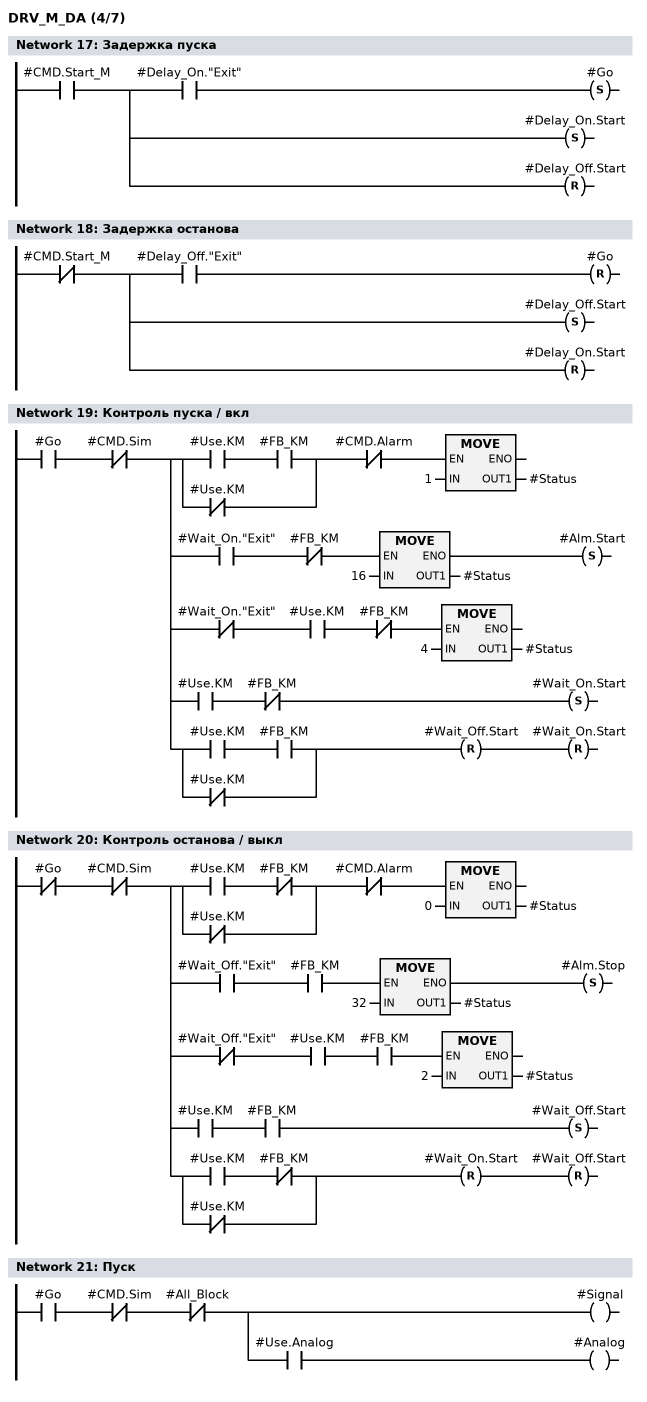
   RUNG wire#powerrail
      Contact( #CMD.Start_M )
      wire#w1
      Contact( #Delay_On."Exit" )
      S_Coil( #Go )
   END_RUNG
   RUNG wire#w1
      S_Coil( #Delay_On.Start )
   END_RUNG
   RUNG wire#w1
      R_Coil( #Delay_Off.Start )
   END_RUNG
   // the same network as SCL:
   IF #CMD.Start_M AND #Delay_On."Exit" THEN #Go := TRUE; END_IF;
   IF #CMD.Start_M THEN
       #Delay_On.Start := TRUE;
       #Delay_Off.Start := FALSE;
   END_IF;
END_REGION

REGION Network 18: Задержка останова
   RUNG wire#powerrail
      I_Contact( #CMD.Start_M )
      wire#w1
      Contact( #Delay_Off."Exit" )
      R_Coil( #Go )
   END_RUNG
   RUNG wire#w1
      S_Coil( #Delay_Off.Start )
   END_RUNG
   RUNG wire#w1
      R_Coil( #Delay_On.Start )
   END_RUNG
   // the same network as SCL:
   IF NOT #CMD.Start_M AND #Delay_Off."Exit" THEN #Go := FALSE; END_IF;
   IF NOT #CMD.Start_M THEN
       #Delay_Off.Start := TRUE;
       #Delay_On.Start := FALSE;
   END_IF;
END_REGION

REGION Network 19: Контроль пуска / вкл
   RUNG wire#powerrail
      Contact( #Go )
      I_Contact( #CMD.Sim )
      wire#w1
      Contact( #Use.KM )
      Contact( #FB_KM )
      wire#w2
      I_Contact( #CMD.Alarm )
      { S7_GenerateENO := "TRUE" } Move(in := 1, out1 => #Status)
   END_RUNG
   RUNG wire#w1
      I_Contact( #Use.KM )
   END_RUNG wire#w2
   RUNG wire#w1
      Contact( #Wait_On."Exit" )
      I_Contact( #FB_KM )
      { S7_GenerateENO := "TRUE" } Move(in := 16, out1 => #Status)
      S_Coil( #Alm.Start )
   END_RUNG
   RUNG wire#w1
      I_Contact( #Wait_On."Exit" )
      Contact( #Use.KM )
      I_Contact( #FB_KM )
      { S7_GenerateENO := "TRUE" } Move(in := 4, out1 => #Status)
   END_RUNG
   RUNG wire#w1
      Contact( #Use.KM )
      I_Contact( #FB_KM )
      S_Coil( #Wait_On.Start )
   END_RUNG
   RUNG wire#w1
      Contact( #Use.KM )
      Contact( #FB_KM )
      wire#w3
      R_Coil( #Wait_Off.Start )
      R_Coil( #Wait_On.Start )
   END_RUNG
   RUNG wire#w1
      I_Contact( #Use.KM )
   END_RUNG wire#w3
   // the same network as SCL:
   // ENO of a box is taken as its EN; it also drops when the box reports an error
   #_w1 := #Go AND NOT #CMD.Sim;
   IF #_w1 AND ((#Use.KM AND #FB_KM) OR NOT #Use.KM) AND NOT #CMD.Alarm THEN #Status := 1; END_IF;
   IF #_w1 AND #Wait_On."Exit" AND NOT #FB_KM THEN
       #Status := 16;
       #Alm.Start := TRUE;
   END_IF;
   IF #_w1 AND NOT #Wait_On."Exit" AND #Use.KM AND NOT #FB_KM THEN #Status := 4; END_IF;
   IF #_w1 AND #Use.KM AND NOT #FB_KM THEN #Wait_On.Start := TRUE; END_IF;
   IF #_w1 AND ((#Use.KM AND #FB_KM) OR NOT #Use.KM) THEN
       #Wait_Off.Start := FALSE;
       #Wait_On.Start := FALSE;
   END_IF;
END_REGION

REGION Network 20: Контроль останова / выкл
   RUNG wire#powerrail
      I_Contact( #Go )
      I_Contact( #CMD.Sim )
      wire#w1
      Contact( #Use.KM )
      I_Contact( #FB_KM )
      wire#w2
      I_Contact( #CMD.Alarm )
      { S7_GenerateENO := "TRUE" } Move(in := 0, out1 => #Status)
   END_RUNG
   RUNG wire#w1
      I_Contact( #Use.KM )
   END_RUNG wire#w2
   RUNG wire#w1
      Contact( #Wait_Off."Exit" )
      Contact( #FB_KM )
      { S7_GenerateENO := "TRUE" } Move(in := 32, out1 => #Status)
      S_Coil( #Alm.Stop )
   END_RUNG
   RUNG wire#w1
      I_Contact( #Wait_Off."Exit" )
      Contact( #Use.KM )
      Contact( #FB_KM )
      { S7_GenerateENO := "TRUE" } Move(in := 2, out1 => #Status)
   END_RUNG
   RUNG wire#w1
      Contact( #Use.KM )
      Contact( #FB_KM )
      S_Coil( #Wait_Off.Start )
   END_RUNG
   RUNG wire#w1
      Contact( #Use.KM )
      I_Contact( #FB_KM )
      wire#w3
      R_Coil( #Wait_On.Start )
      R_Coil( #Wait_Off.Start )
   END_RUNG
   RUNG wire#w1
      I_Contact( #Use.KM )
   END_RUNG wire#w3
   // the same network as SCL:
   // ENO of a box is taken as its EN; it also drops when the box reports an error
   #_w1 := NOT #Go AND NOT #CMD.Sim;
   IF #_w1 AND ((#Use.KM AND NOT #FB_KM) OR NOT #Use.KM) AND NOT #CMD.Alarm THEN #Status := 0; END_IF;
   IF #_w1 AND #Wait_Off."Exit" AND #FB_KM THEN
       #Status := 32;
       #Alm.Stop := TRUE;
   END_IF;
   IF #_w1 AND NOT #Wait_Off."Exit" AND #Use.KM AND #FB_KM THEN #Status := 2; END_IF;
   IF #_w1 AND #Use.KM AND #FB_KM THEN #Wait_Off.Start := TRUE; END_IF;
   IF #_w1 AND ((#Use.KM AND NOT #FB_KM) OR NOT #Use.KM) THEN
       #Wait_On.Start := FALSE;
       #Wait_Off.Start := FALSE;
   END_IF;
END_REGION

REGION Network 21: Пуск
   RUNG wire#powerrail
      Contact( #Go )
      I_Contact( #CMD.Sim )
      I_Contact( #All_Block )
      wire#w1
      Coil( #Signal )
   END_RUNG
   RUNG wire#w1
      Contact( #Use.Analog )
      Coil( #Analog )
   END_RUNG
   // the same network as SCL:
   #Signal := #Go AND NOT #CMD.Sim AND NOT #All_Block;
   #Analog := #Signal AND #Use.Analog;
END_REGION

REGION Network 22: Сервисный режим
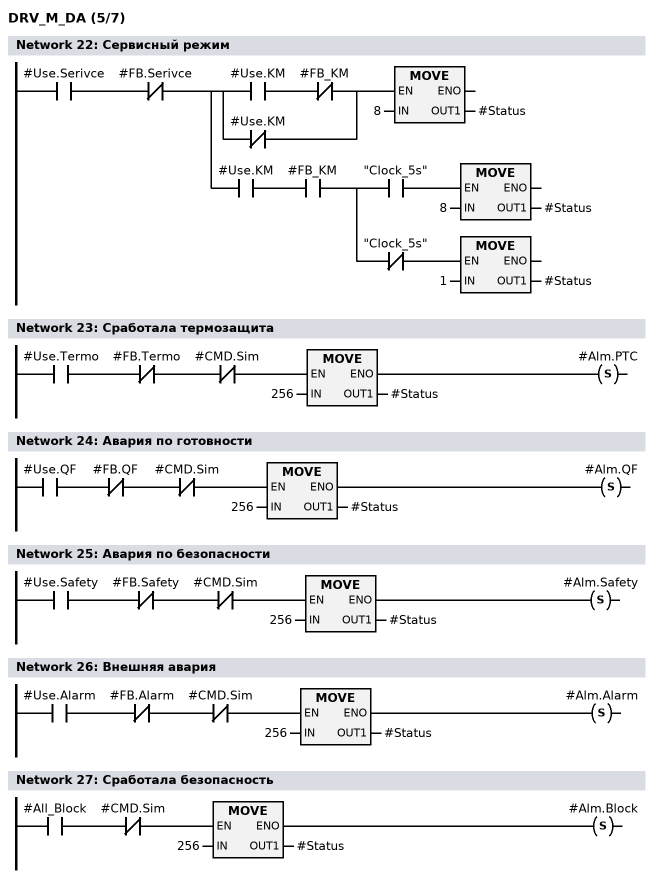
   RUNG wire#powerrail
      Contact( #Use.Serivce )
      I_Contact( #FB.Serivce )
      wire#w1
      Contact( #Use.KM )
      I_Contact( #FB_KM )
      wire#w2
      Move(in := 8, out1 => #Status)
   END_RUNG
   RUNG wire#w1
      I_Contact( #Use.KM )
   END_RUNG wire#w2
   RUNG wire#w1
      Contact( #Use.KM )
      Contact( #FB_KM )
      wire#w3
      Contact( "Clock_5s" )
      Move(in := 8, out1 => #Status)
   END_RUNG
   RUNG wire#w3
      I_Contact( "Clock_5s" )
      Move(in := 1, out1 => #Status)
   END_RUNG
   // the same network as SCL:
   #_w1 := #Use.Serivce AND NOT #FB.Serivce;
   IF #_w1 AND ((#Use.KM AND NOT #FB_KM) OR NOT #Use.KM) THEN #Status := 8; END_IF;
   #_w2 := #_w1 AND #Use.KM AND #FB_KM;
   IF #_w2 AND "Clock_5s" THEN #Status := 8; END_IF;
   IF #_w2 AND NOT "Clock_5s" THEN #Status := 1; END_IF;
END_REGION

REGION Network 23: Сработала термозащита
   RUNG wire#powerrail
      Contact( #Use.Termo )
      I_Contact( #FB.Termo )
      I_Contact( #CMD.Sim )
      { S7_GenerateENO := "TRUE" } Move(in := 256, out1 => #Status)
      S_Coil( #Alm.PTC )
   END_RUNG
   // the same network as SCL:
   // ENO of a box is taken as its EN; it also drops when the box reports an error
   IF #Use.Termo AND NOT #FB.Termo AND NOT #CMD.Sim THEN
       #Status := 256;
       #Alm.PTC := TRUE;
   END_IF;
END_REGION

REGION Network 24: Авария по готовности
   RUNG wire#powerrail
      Contact( #Use.QF )
      I_Contact( #FB.QF )
      I_Contact( #CMD.Sim )
      { S7_GenerateENO := "TRUE" } Move(in := 256, out1 => #Status)
      S_Coil( #Alm.QF )
   END_RUNG
   // the same network as SCL:
   // ENO of a box is taken as its EN; it also drops when the box reports an error
   IF #Use.QF AND NOT #FB.QF AND NOT #CMD.Sim THEN
       #Status := 256;
       #Alm.QF := TRUE;
   END_IF;
END_REGION

REGION Network 25: Авария по безопасности
   RUNG wire#powerrail
      Contact( #Use.Safety )
      I_Contact( #FB.Safety )
      I_Contact( #CMD.Sim )
      { S7_GenerateENO := "TRUE" } Move(in := 256, out1 => #Status)
      S_Coil( #Alm.Safety )
   END_RUNG
   // the same network as SCL:
   // ENO of a box is taken as its EN; it also drops when the box reports an error
   IF #Use.Safety AND NOT #FB.Safety AND NOT #CMD.Sim THEN
       #Status := 256;
       #Alm.Safety := TRUE;
   END_IF;
END_REGION

REGION Network 26: Внешняя авария
   RUNG wire#powerrail
      Contact( #Use.Alarm )
      I_Contact( #FB.Alarm )
      I_Contact( #CMD.Sim )
      { S7_GenerateENO := "TRUE" } Move(in := 256, out1 => #Status)
      S_Coil( #Alm.Alarm )
   END_RUNG
   // the same network as SCL:
   // ENO of a box is taken as its EN; it also drops when the box reports an error
   IF #Use.Alarm AND NOT #FB.Alarm AND NOT #CMD.Sim THEN
       #Status := 256;
       #Alm.Alarm := TRUE;
   END_IF;
END_REGION

REGION Network 27: Сработала безопасность
   RUNG wire#powerrail
      Contact( #All_Block )
      I_Contact( #CMD.Sim )
      { S7_GenerateENO := "TRUE" } Move(in := 256, out1 => #Status)
      S_Coil( #Alm.Block )
   END_RUNG
   // the same network as SCL:
   // ENO of a box is taken as its EN; it also drops when the box reports an error
   IF #All_Block AND NOT #CMD.Sim THEN
       #Status := 256;
       #Alm.Block := TRUE;
   END_IF;
END_REGION

REGION Network 28: Сигнал аварии
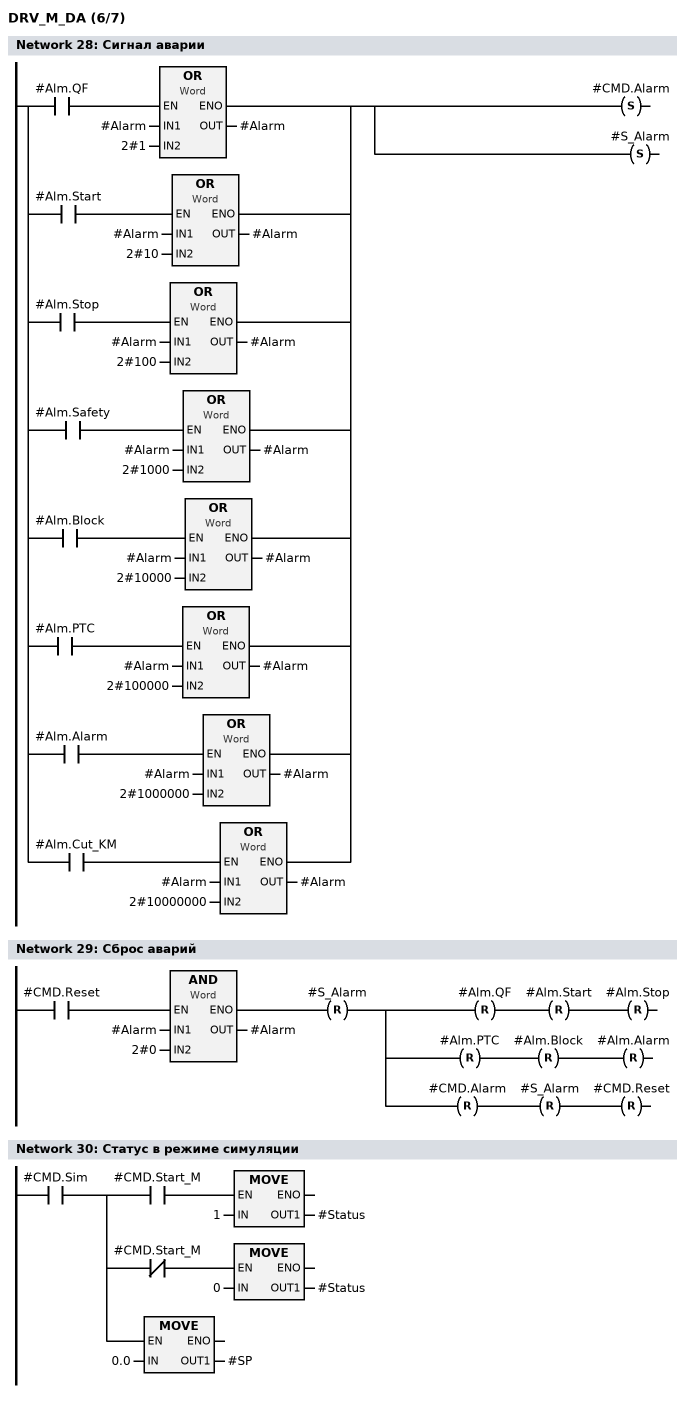
   // no checked SCL form for this network; see the picture
END_REGION

REGION Network 29: Сброс аварий
   // no checked SCL form for this network; see the picture
END_REGION

REGION Network 30: Статус в режиме симуляции
   RUNG wire#powerrail
      Contact( #CMD.Sim )
      wire#w1
      Contact( #CMD.Start_M )
      { S7_GenerateENO := "TRUE" } Move(in := 1, out1 => #Status)
   END_RUNG
   RUNG wire#w1
      I_Contact( #CMD.Start_M )
      { S7_GenerateENO := "TRUE" } Move(in := 0, out1 => #Status)
   END_RUNG
   RUNG wire#w1
      Move(in := 0.0, out1 => #SP)
   END_RUNG
   // the same network as SCL:
   IF #CMD.Sim AND #CMD.Start_M THEN #Status := 1; END_IF;
   IF #CMD.Sim AND NOT #CMD.Start_M THEN #Status := 0; END_IF;
   IF #CMD.Sim THEN #SP := 0.0; END_IF;
END_REGION

REGION Network 31: Статус в локальным режиме
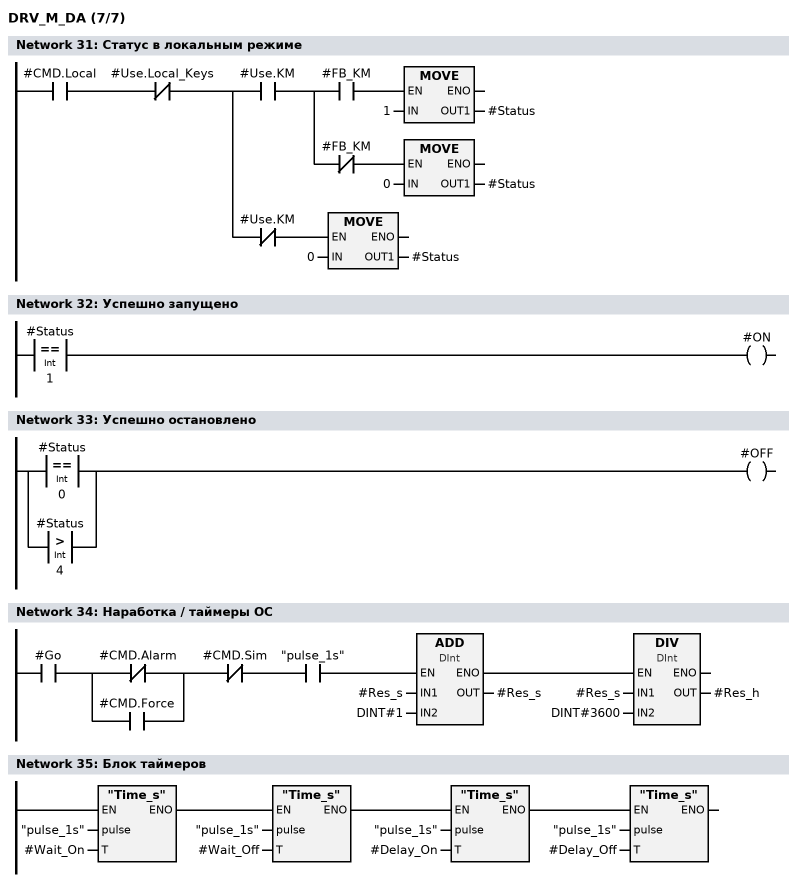
   RUNG wire#powerrail
      Contact( #CMD.Local )
      I_Contact( #Use.Local_Keys )
      wire#w1
      Contact( #Use.KM )
      wire#w2
      Contact( #FB_KM )
      { S7_GenerateENO := "TRUE" } Move(in := 1, out1 => #Status)
   END_RUNG
   RUNG wire#w2
      I_Contact( #FB_KM )
      { S7_GenerateENO := "TRUE" } Move(in := 0, out1 => #Status)
   END_RUNG
   RUNG wire#w1
      I_Contact( #Use.KM )
      { S7_GenerateENO := "TRUE" } Move(in := 0, out1 => #Status)
   END_RUNG
   // the same network as SCL:
   #_w1 := #CMD.Local AND NOT #Use.Local_Keys;
   #_w2 := #_w1 AND #Use.KM;
   IF #_w2 AND #FB_KM THEN #Status := 1; END_IF;
   IF #_w2 AND NOT #FB_KM THEN #Status := 0; END_IF;
   IF #_w1 AND NOT #Use.KM THEN #Status := 0; END_IF;
END_REGION

REGION Network 32: Успешно запущено
   RUNG wire#powerrail
      { S7_Templates := "SrcType := Int" } EQ_Contact(in1 := #Status, in2 := 1)
      Coil( #ON )
   END_RUNG
   // the same network as SCL:
   #ON := #Status = 1;
END_REGION

REGION Network 33: Успешно остановлено
   RUNG wire#powerrail
      { S7_Templates := "SrcType := Int" } EQ_Contact(in1 := #Status, in2 := 0)
      wire#w1
      Coil( #OFF )
   END_RUNG
   RUNG wire#powerrail
      { S7_Templates := "SrcType := Int" } GT_Contact(in1 := #Status, in2 := 4)
   END_RUNG wire#w1
   // the same network as SCL:
   #OFF := (#Status = 0) OR (#Status > 4);
END_REGION

REGION Network 34: Наработка / таймеры ОС
   RUNG wire#powerrail
      Contact( #Go )
      wire#w1
      I_Contact( #CMD.Alarm )
      wire#w2
      I_Contact( #CMD.Sim )
      Contact( "pulse_1s" )
      { S7_Templates := "SrcType := DInt"; S7_GenerateENO := "TRUE" } Add(in1 := #Res_s, in2 := DINT#1, out => #Res_s)
      { S7_Templates := "SrcType := DInt"; S7_GenerateENO := "TRUE" } Div(in1 := #Res_s, in2 := DINT#3600, out => #Res_h)
   END_RUNG
   RUNG wire#w1
      Contact( #CMD.Force )
   END_RUNG wire#w2
   // the same network as SCL:
   // ENO of a box is taken as its EN; it also drops when the box reports an error
   IF #Go AND (NOT #CMD.Alarm OR #CMD.Force) AND NOT #CMD.Sim AND "pulse_1s" THEN
       #Res_s := #Res_s + DINT#1;
       #Res_h := #Res_s / DINT#3600;
   END_IF;
END_REGION

REGION Network 35: Блок таймеров
   RUNG wire#powerrail
      "Time_s"(pulse := "pulse_1s", T := #Wait_On)
      "Time_s"(pulse := "pulse_1s", T := #Wait_Off)
      "Time_s"(pulse := "pulse_1s", T := #Delay_On)
      "Time_s"(pulse := "pulse_1s", T := #Delay_Off)
   END_RUNG
   // the same network as SCL:
   "Time_s"(pulse := "pulse_1s", T := #Wait_On, ENO => #_w1);
   "Time_s"(EN := #_w1, pulse := "pulse_1s", T := #Wait_Off, ENO => #_w2);
   "Time_s"(EN := #_w2, pulse := "pulse_1s", T := #Delay_On, ENO => #_w3);
   IF #_w3 THEN "Time_s"(pulse := "pulse_1s", T := #Delay_Off); END_IF;
END_REGION
END_FUNCTION_BLOCK

FUNCTION_BLOCK "DRV_V_D2"   // FB112, LAD
{ S7_Optimized_Access := 'FALSE' }
VERSION : 0.1
   VAR_INPUT
      FB_QF : Bool;   // защитный автомат / Защитный автомат
      FB_KM_Open : Bool;   // Пускатель - открыть
      FB_KM_Close : Bool;   // Пускатель - закрыть
      FB_Service : Bool;   // авария частотника / Сервисный выключатель
      FB_Open : Bool;   // ОС - открыто
      FB_Close : Bool;   // ОС - закрыто
      Local_Open : Bool;   // Локальное открытие
      Local_Close : Bool;   // Локальное закрытие
      All_Block : Bool;   // Аварийный останов
   END_VAR
   VAR_OUTPUT
      CMD_Open : Bool;   // Команда - открыть
      CMD_Close : Bool;   // Команда - закрыть
   END_VAR
   VAR_IN_OUT
      S_Alarm : Bool;   // Наличие аварии
   END_VAR
   VAR
      CMD : Struct   // Основные команды / Блок команд
         Hand : Bool;   // 0 - авто, 1 - ручной / 0 - Авто, 1 - Ручной
         Start_A : Bool;   // Автозапуск / Запуск в авторежиме
         Start_M : Bool;   // Ручной - вперёд / Запуск в ручном режиме
         Force : Bool;   // Принудительный
         Lock : Bool;   // Блокировать / Блокировка
         Local : Bool;   // Локальный
         Service : Bool;   // Сервис
         Safety : Bool;   // Безопасность
         Alarm : Bool;   // Есть авария / Авария
         Reset : Bool;   // Сброс аварий
         Sim : Bool;   // Режим симуляции
      END_STRUCT;
      Mode : Int;   // Режим работы
      Status : Int;   // Статус устройства
      Use : Struct   // Функционал
         Ready : Bool := true;   // Готовность
         QF : Bool := true;   // Защитный автомат
         KM_Open : Bool := true;   // Пускатель - открыть
         KM_Close : Bool;   // Пускатель - закрыть
         Serivce : Bool;   // Сервисный выключатель
         Open : Bool := true;   // ОС - открыто
         Close : Bool;   // ОС - закрыто
         Local_Keys : Bool;   // Использовать локальное управление
         One_KM : Bool;   // Общий пускатель
         Electro : Bool;   // Электропривод
      END_STRUCT;
      FB : Struct   // Функционал
         Ready : Bool;   // Готовность к запуску
         QF : Bool;   // Защитный автомат
         KM_Open : Bool;   // Пускатель - открыть
         KM_Close : Bool;   // Пускатель - закрыть
         Serivce : Bool;   // Сервисный выключатель
         Open : Bool;   // ОС - открыто
         Close : Bool;   // ОС - закрыто
         Reserv : Bool;
         Local_Open : Bool;   // Локальное открытие
         Local_Close : Bool;   // Локальное закрытие
      END_STRUCT;
      Go : Bool;   // Запуск
      ON : Bool;   // Успешно запущено
      OFF : Bool;   // Успешно остановлено
      G_Sim_On : Bool;   // Глобальная симуляция - начать
      G_Sim_Off : Bool;   // Глобальная симуляция - завершить
      REQ_Open : Bool;   // Запрос на открытие
      REQ_Close : Bool;   // Запрос на закрытие
      Wait_On : Struct   // Ожидание ОС контактора / Время на запуск
         SP : Int := 4;
         Now : Int;
         "Exit" : Bool;
         Start : Bool;
         Pause : Bool;
         Reset : Bool;   // Сброс таймера
      END_STRUCT;
      Wait_Off : Struct   // Ожидание концевиков / Время на останов
         SP : Int := 4;
         Now : Int;
         "Exit" : Bool;
         Start : Bool;
         Pause : Bool;
         Reset : Bool;   // Сброс таймера
      END_STRUCT;
      Delay_On : Struct
         SP : Real;   // Уставка
         Now : Real;   // Текущий счёт
         One : Real := 0.1;   // Вес импульса
         Progress : Real;   // Прогресс выполнения
         "Exit" : Bool;   // Счёт завершён
         Start : Bool;   // Запуск
         Pause : Bool;   // Пауза
         Reset : Bool;   // Сброс счёта
         pos : Bool;   // Контроль фронта сигнала
      END_STRUCT;
      Delay_Off : Struct
         SP : Real;   // Уставка
         Now : Real;   // Текущий счёт
         One : Real := 0.1;   // Вес импульса
         Progress : Real;   // Прогресс выполнения
         "Exit" : Bool;   // Счёт завершён
         Start : Bool;   // Запуск
         Pause : Bool;   // Пауза
         Reset : Bool;   // Сброс счёта
         pos : Bool;   // Контроль фронта сигнала
      END_STRUCT;
      Inv : Struct   // Инверсия сигналов
         Reserv : Bool;
         QF : Bool;   // Защитный автомат
         KM_Open : Bool;   // Пускатель - открыть
         KM_Close : Bool;   // Пускатель - закрыть
         Serivce : Bool;   // Сервисный выключатель
         Open : Bool;   // ОС - открыто
         Close : Bool;   // ОС - закрыто
         CMD : Bool;   // Инверсия управляющих сигналов
         Local_Open : Bool;   // Локальное открытие
         Local_Close : Bool;   // Локальное закрытие
      END_STRUCT;
      Alm : Struct   // Сбор аварий / Список аварий
         Block : Bool;   // Аварийная остановка
         QF : Bool;   // привод не готов / Выбило защитный автомат
         KM_Open : Bool;   // Не сработал пускатель - открыть
         KM_Close : Bool;   // Не сработал пускатель - закрыть
         Two_S : Bool;   // Две ОС
         Open : Bool;   // Не сработал концевик - открыто
         Close : Bool;   // термозащита / Не сработал концевик - закрыто
      END_STRUCT;
      Alarm : Word;   // Слово аварий
      Res_h : DInt;   // наработка (ч)
      Res_s : DInt;   // наработка (с)
      REQ_ON : "DRV_Micro";   // Контроль пускателя на открытие
      REQ_OFF : "DRV_Micro";   // Контроль пускателя на закрытие
   END_VAR
   VAR_TEMP   // added for the SCL form of the ladder/FBD networks
      _w1 : Bool;
      _w2 : Bool;
      _w3 : Bool;
   END_VAR
BEGIN

REGION Network 1: Режим глобальной симуляции
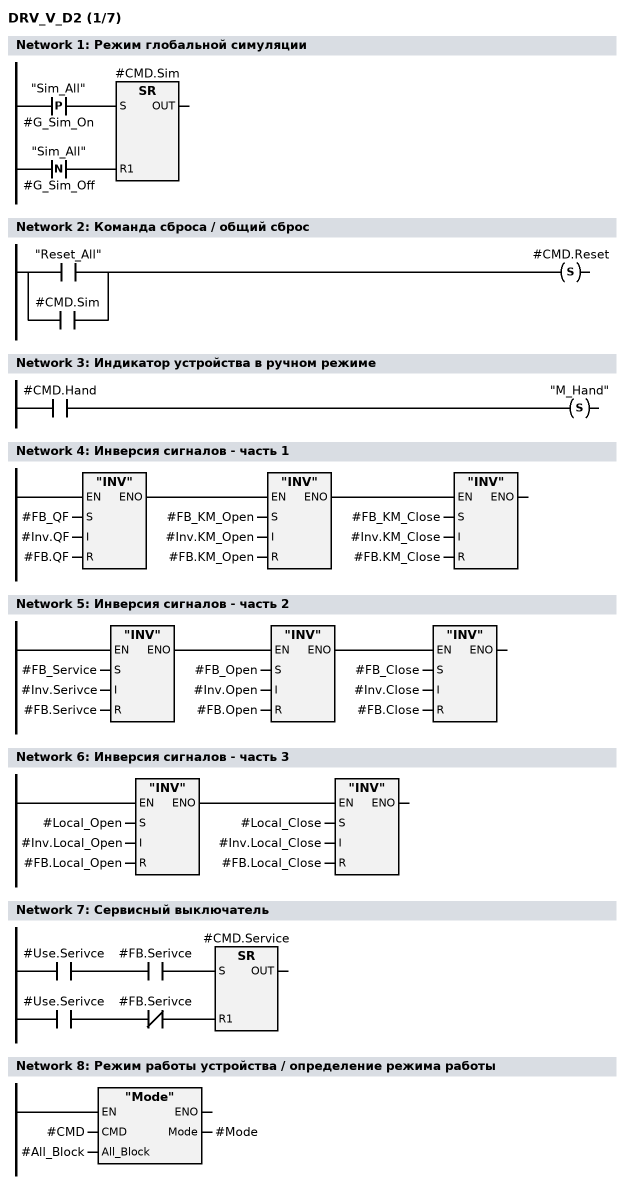
   RUNG wire#powerrail
      P_Contact(operand := "Sim_All", bit := #G_Sim_On)
      S_SR(operand := #CMD.Sim, r1 := wire#w1)
   END_RUNG
   RUNG wire#powerrail
      N_Contact(operand := "Sim_All", bit := #G_Sim_Off)
   END_RUNG wire#w1
   // the same network as SCL:
   #_w1 := "Sim_All" AND NOT #G_Sim_On;   // rising edge of "Sim_All"
   #G_Sim_On := "Sim_All";
   #_w2 := NOT "Sim_All" AND #G_Sim_Off;   // falling edge of "Sim_All"
   #G_Sim_Off := "Sim_All";
   IF #_w1 THEN
       #CMD.Sim := TRUE;   // SR flip-flop
   END_IF;
   IF #_w2 THEN #CMD.Sim := FALSE; END_IF;
END_REGION

REGION Network 2: Команда сброса / общий сброс
   RUNG wire#powerrail
      Contact( "Reset_All" )
      wire#w1
      S_Coil( #CMD.Reset )
   END_RUNG
   RUNG wire#powerrail
      Contact( #CMD.Sim )
   END_RUNG wire#w1
   // the same network as SCL:
   IF "Reset_All" OR #CMD.Sim THEN #CMD.Reset := TRUE; END_IF;
END_REGION

REGION Network 3: Индикатор устройства в ручном режиме
   RUNG wire#powerrail
      Contact( #CMD.Hand )
      S_Coil( "M_Hand" )
   END_RUNG
   // the same network as SCL:
   IF #CMD.Hand THEN "M_Hand" := TRUE; END_IF;
END_REGION

REGION Network 4: Инверсия сигналов - часть 1
   RUNG wire#powerrail
      "INV"(S := #FB_QF, I := #Inv.QF, R := #FB.QF)
      "INV"(S := #FB_KM_Open, I := #Inv.KM_Open, R := #FB.KM_Open)
      "INV"(S := #FB_KM_Close, I := #Inv.KM_Close, R := #FB.KM_Close)
   END_RUNG
   // the same network as SCL:
   "INV"(S := #FB_QF, I := #Inv.QF, R := #FB.QF, ENO => #_w1);
   "INV"(EN := #_w1, S := #FB_KM_Open, I := #Inv.KM_Open, R := #FB.KM_Open, ENO => #_w2);
   IF #_w2 THEN "INV"(S := #FB_KM_Close, I := #Inv.KM_Close, R := #FB.KM_Close); END_IF;
END_REGION

REGION Network 5: Инверсия сигналов - часть 2
   RUNG wire#powerrail
      "INV"(S := #FB_Service, I := #Inv.Serivce, R := #FB.Serivce)
      "INV"(S := #FB_Open, I := #Inv.Open, R := #FB.Open)
      "INV"(S := #FB_Close, I := #Inv.Close, R := #FB.Close)
   END_RUNG
   // the same network as SCL:
   "INV"(S := #FB_Service, I := #Inv.Serivce, R := #FB.Serivce, ENO => #_w1);
   "INV"(EN := #_w1, S := #FB_Open, I := #Inv.Open, R := #FB.Open, ENO => #_w2);
   IF #_w2 THEN "INV"(S := #FB_Close, I := #Inv.Close, R := #FB.Close); END_IF;
END_REGION

REGION Network 6: Инверсия сигналов - часть 3
   RUNG wire#powerrail
      "INV"(S := #Local_Open, I := #Inv.Local_Open, R := #FB.Local_Open)
      "INV"(S := #Local_Close, I := #Inv.Local_Close, R := #FB.Local_Close)
   END_RUNG
   // the same network as SCL:
   "INV"(S := #Local_Open, I := #Inv.Local_Open, R := #FB.Local_Open, ENO => #_w1);
   IF #_w1 THEN "INV"(S := #Local_Close, I := #Inv.Local_Close, R := #FB.Local_Close); END_IF;
END_REGION

REGION Network 7: Сервисный выключатель
   RUNG wire#powerrail
      Contact( #Use.Serivce )
      Contact( #FB.Serivce )
      S_SR(operand := #CMD.Service, r1 := wire#w1)
   END_RUNG
   RUNG wire#powerrail
      Contact( #Use.Serivce )
      I_Contact( #FB.Serivce )
   END_RUNG wire#w1
   // the same network as SCL:
   IF #Use.Serivce AND #FB.Serivce THEN
       #CMD.Service := TRUE;   // SR flip-flop
   END_IF;
   IF #Use.Serivce AND NOT #FB.Serivce THEN #CMD.Service := FALSE; END_IF;
END_REGION

REGION Network 8: Режим работы устройства / определение режима работы
   RUNG wire#powerrail
      "Mode"(CMD := #CMD, All_Block := #All_Block, Mode => #Mode)
   END_RUNG
   // the same network as SCL:
   "Mode"(CMD := #CMD, All_Block := #All_Block, Mode => #Mode);
END_REGION

REGION Network 9: Готовность к запуску
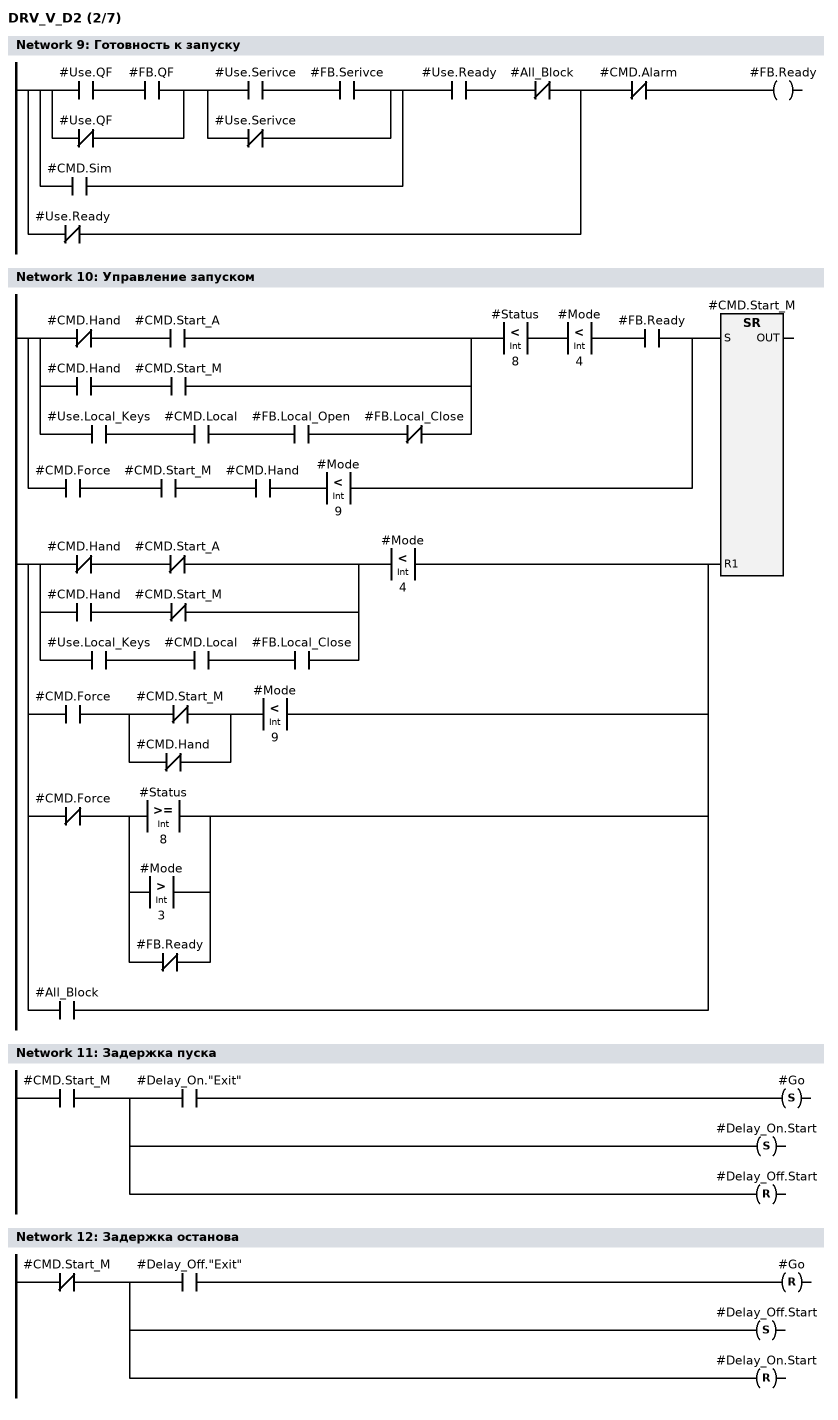
   RUNG wire#powerrail
      Contact( #Use.QF )
      Contact( #FB.QF )
      wire#w1
      Contact( #Use.Serivce )
      Contact( #FB.Serivce )
      wire#w2
      Contact( #Use.Ready )
      I_Contact( #All_Block )
      wire#w3
      I_Contact( #CMD.Alarm )
      Coil( #FB.Ready )
   END_RUNG
   RUNG wire#powerrail
      I_Contact( #Use.QF )
   END_RUNG wire#w1
   RUNG wire#w1
      I_Contact( #Use.Serivce )
   END_RUNG wire#w2
   RUNG wire#powerrail
      Contact( #CMD.Sim )
   END_RUNG wire#w2
   RUNG wire#powerrail
      I_Contact( #Use.Ready )
   END_RUNG wire#w3
   // the same network as SCL:
   #FB.Ready := ((((((#Use.QF AND #FB.QF) OR NOT #Use.QF) AND ((#Use.Serivce AND #FB.Serivce) OR NOT #Use.Serivce)) OR #CMD.Sim) AND #Use.Ready AND NOT #All_Block) OR NOT #Use.Ready) AND NOT #CMD.Alarm;
END_REGION

REGION Network 10: Управление запуском
   RUNG wire#powerrail
      I_Contact( #CMD.Hand )
      Contact( #CMD.Start_A )
      wire#w1
      { S7_Templates := "SrcType := Int" } LT_Contact(in1 := #Status, in2 := 8)
      { S7_Templates := "SrcType := Int" } LT_Contact(in1 := #Mode, in2 := 4)
      Contact( #FB.Ready )
      wire#w2
      S_SR(operand := #CMD.Start_M, r1 := wire#w7)
   END_RUNG
   RUNG wire#powerrail
      Contact( #CMD.Hand )
      Contact( #CMD.Start_M )
   END_RUNG wire#w1
   RUNG wire#powerrail
      Contact( #Use.Local_Keys )
      Contact( #CMD.Local )
      Contact( #FB.Local_Open )
      I_Contact( #FB.Local_Close )
   END_RUNG wire#w1
   RUNG wire#powerrail
      Contact( #CMD.Force )
      Contact( #CMD.Start_M )
      Contact( #CMD.Hand )
      { S7_Templates := "SrcType := Int" } LT_Contact(in1 := #Mode, in2 := 9)
   END_RUNG wire#w2
   RUNG wire#powerrail
      I_Contact( #CMD.Hand )
      I_Contact( #CMD.Start_A )
      wire#w3
      { S7_Templates := "SrcType := Int" } LT_Contact(in1 := #Mode, in2 := 4)
   END_RUNG wire#w7
   RUNG wire#powerrail
      Contact( #CMD.Hand )
      I_Contact( #CMD.Start_M )
   END_RUNG wire#w3
   RUNG wire#powerrail
      Contact( #Use.Local_Keys )
      Contact( #CMD.Local )
      Contact( #FB.Local_Close )
   END_RUNG wire#w3
   RUNG wire#powerrail
      Contact( #CMD.Force )
      wire#w4
      I_Contact( #CMD.Start_M )
      wire#w5
      { S7_Templates := "SrcType := Int" } LT_Contact(in1 := #Mode, in2 := 9)
   END_RUNG wire#w7
   RUNG wire#w4
      I_Contact( #CMD.Hand )
   END_RUNG wire#w5
   RUNG wire#powerrail
      I_Contact( #CMD.Force )
      wire#w6
      { S7_Templates := "SrcType := Int" } GE_Contact(in1 := #Status, in2 := 8)
   END_RUNG wire#w7
   RUNG wire#w6
      { S7_Templates := "SrcType := Int" } GT_Contact(in1 := #Mode, in2 := 3)
   END_RUNG wire#w7
   RUNG wire#w6
      I_Contact( #FB.Ready )
   END_RUNG wire#w7
   RUNG wire#powerrail
      Contact( #All_Block )
   END_RUNG wire#w7
   // the same network as SCL:
   #_w1 := (((NOT #CMD.Hand AND NOT #CMD.Start_A) OR (#CMD.Hand AND NOT #CMD.Start_M) OR (#Use.Local_Keys AND #CMD.Local AND #FB.Local_Close)) AND (#Mode < 4)) OR (#CMD.Force AND (NOT #CMD.Start_M OR NOT #CMD.Hand) AND (#Mode < 9)) OR (NOT #CMD.Force AND ((#Status >= 8) OR (#Mode > 3) OR NOT #FB.Ready)) OR #All_Block;
   IF (((NOT #CMD.Hand AND #CMD.Start_A) OR (#CMD.Hand AND #CMD.Start_M) OR (#Use.Local_Keys AND #CMD.Local AND #FB.Local_Open AND NOT #FB.Local_Close)) AND (#Status < 8) AND (#Mode < 4) AND #FB.Ready) OR (#CMD.Force AND #CMD.Start_M AND #CMD.Hand AND (#Mode < 9)) THEN
       #CMD.Start_M := TRUE;   // SR flip-flop
   END_IF;
   IF #_w1 THEN #CMD.Start_M := FALSE; END_IF;
END_REGION

REGION Network 11: Задержка пуска
   RUNG wire#powerrail
      Contact( #CMD.Start_M )
      wire#w1
      Contact( #Delay_On."Exit" )
      S_Coil( #Go )
   END_RUNG
   RUNG wire#w1
      S_Coil( #Delay_On.Start )
   END_RUNG
   RUNG wire#w1
      R_Coil( #Delay_Off.Start )
   END_RUNG
   // the same network as SCL:
   IF #CMD.Start_M AND #Delay_On."Exit" THEN #Go := TRUE; END_IF;
   IF #CMD.Start_M THEN
       #Delay_On.Start := TRUE;
       #Delay_Off.Start := FALSE;
   END_IF;
END_REGION

REGION Network 12: Задержка останова
   RUNG wire#powerrail
      I_Contact( #CMD.Start_M )
      wire#w1
      Contact( #Delay_Off."Exit" )
      R_Coil( #Go )
   END_RUNG
   RUNG wire#w1
      S_Coil( #Delay_Off.Start )
   END_RUNG
   RUNG wire#w1
      R_Coil( #Delay_On.Start )
   END_RUNG
   // the same network as SCL:
   IF NOT #CMD.Start_M AND #Delay_Off."Exit" THEN #Go := FALSE; END_IF;
   IF NOT #CMD.Start_M THEN
       #Delay_Off.Start := TRUE;
       #Delay_On.Start := FALSE;
   END_IF;
END_REGION

REGION Network 13: Команда открытия / выкл
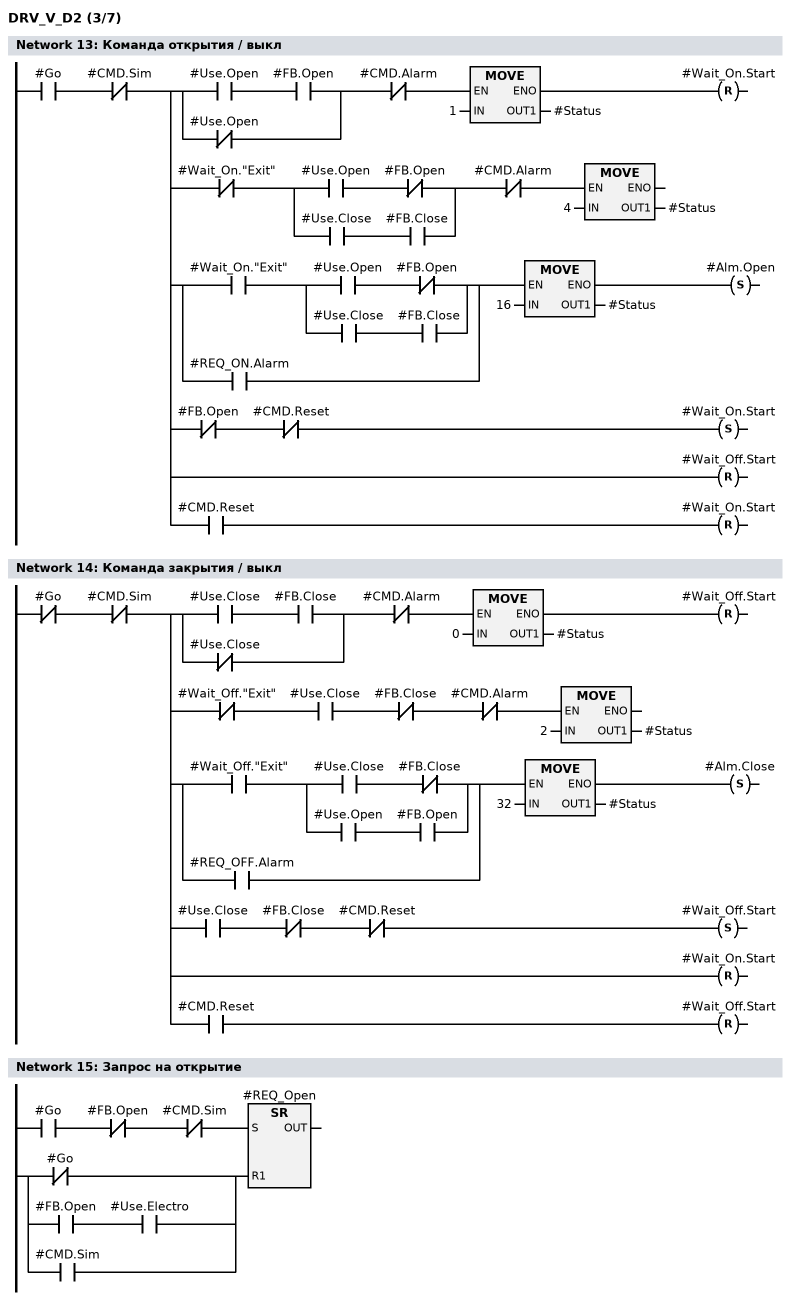
   RUNG wire#powerrail
      Contact( #Go )
      I_Contact( #CMD.Sim )
      wire#w1
      Contact( #Use.Open )
      Contact( #FB.Open )
      wire#w2
      I_Contact( #CMD.Alarm )
      { S7_GenerateENO := "TRUE" } Move(in := 1, out1 => #Status)
      R_Coil( #Wait_On.Start )
   END_RUNG
   RUNG wire#w1
      I_Contact( #Use.Open )
   END_RUNG wire#w2
   RUNG wire#w1
      I_Contact( #Wait_On."Exit" )
      wire#w3
      Contact( #Use.Open )
      I_Contact( #FB.Open )
      wire#w4
      I_Contact( #CMD.Alarm )
      { S7_GenerateENO := "TRUE" } Move(in := 4, out1 => #Status)
   END_RUNG
   RUNG wire#w3
      Contact( #Use.Close )
      Contact( #FB.Close )
   END_RUNG wire#w4
   RUNG wire#w1
      Contact( #Wait_On."Exit" )
      wire#w5
      Contact( #Use.Open )
      I_Contact( #FB.Open )
      wire#w6
      { S7_GenerateENO := "TRUE" } Move(in := 16, out1 => #Status)
      S_Coil( #Alm.Open )
   END_RUNG
   RUNG wire#w5
      Contact( #Use.Close )
      Contact( #FB.Close )
   END_RUNG wire#w6
   RUNG wire#w1
      Contact( #REQ_ON.Alarm )
   END_RUNG wire#w6
   RUNG wire#w1
      I_Contact( #FB.Open )
      I_Contact( #CMD.Reset )
      S_Coil( #Wait_On.Start )
   END_RUNG
   RUNG wire#w1
      R_Coil( #Wait_Off.Start )
   END_RUNG
   RUNG wire#w1
      Contact( #CMD.Reset )
      R_Coil( #Wait_On.Start )
   END_RUNG
   // the same network as SCL:
   // ENO of a box is taken as its EN; it also drops when the box reports an error
   #_w1 := #Go AND NOT #CMD.Sim;
   IF #_w1 AND ((#Use.Open AND #FB.Open) OR NOT #Use.Open) AND NOT #CMD.Alarm THEN
       #Status := 1;
       #Wait_On.Start := FALSE;
   END_IF;
   IF #_w1 AND NOT #Wait_On."Exit" AND ((#Use.Open AND NOT #FB.Open) OR (#Use.Close AND #FB.Close)) AND NOT #CMD.Alarm THEN
       #Status := 4;
   END_IF;
   IF #_w1 AND ((#Wait_On."Exit" AND ((#Use.Open AND NOT #FB.Open) OR (#Use.Close AND #FB.Close))) OR #REQ_ON.Alarm) THEN
       #Status := 16;
       #Alm.Open := TRUE;
   END_IF;
   IF #_w1 AND NOT #FB.Open AND NOT #CMD.Reset THEN #Wait_On.Start := TRUE; END_IF;
   IF #_w1 THEN #Wait_Off.Start := FALSE; END_IF;
   IF #_w1 AND #CMD.Reset THEN #Wait_On.Start := FALSE; END_IF;
END_REGION

REGION Network 14: Команда закрытия / выкл
   RUNG wire#powerrail
      I_Contact( #Go )
      I_Contact( #CMD.Sim )
      wire#w1
      Contact( #Use.Close )
      Contact( #FB.Close )
      wire#w2
      I_Contact( #CMD.Alarm )
      { S7_GenerateENO := "TRUE" } Move(in := 0, out1 => #Status)
      R_Coil( #Wait_Off.Start )
   END_RUNG
   RUNG wire#w1
      I_Contact( #Use.Close )
   END_RUNG wire#w2
   RUNG wire#w1
      I_Contact( #Wait_Off."Exit" )
      Contact( #Use.Close )
      I_Contact( #FB.Close )
      I_Contact( #CMD.Alarm )
      { S7_GenerateENO := "TRUE" } Move(in := 2, out1 => #Status)
   END_RUNG
   RUNG wire#w1
      Contact( #Wait_Off."Exit" )
      wire#w3
      Contact( #Use.Close )
      I_Contact( #FB.Close )
      wire#w4
      { S7_GenerateENO := "TRUE" } Move(in := 32, out1 => #Status)
      S_Coil( #Alm.Close )
   END_RUNG
   RUNG wire#w3
      Contact( #Use.Open )
      Contact( #FB.Open )
   END_RUNG wire#w4
   RUNG wire#w1
      Contact( #REQ_OFF.Alarm )
   END_RUNG wire#w4
   RUNG wire#w1
      Contact( #Use.Close )
      I_Contact( #FB.Close )
      I_Contact( #CMD.Reset )
      S_Coil( #Wait_Off.Start )
   END_RUNG
   RUNG wire#w1
      R_Coil( #Wait_On.Start )
   END_RUNG
   RUNG wire#w1
      Contact( #CMD.Reset )
      R_Coil( #Wait_Off.Start )
   END_RUNG
   // the same network as SCL:
   // ENO of a box is taken as its EN; it also drops when the box reports an error
   #_w1 := NOT #Go AND NOT #CMD.Sim;
   IF #_w1 AND ((#Use.Close AND #FB.Close) OR NOT #Use.Close) AND NOT #CMD.Alarm THEN
       #Status := 0;
       #Wait_Off.Start := FALSE;
   END_IF;
   IF #_w1 AND NOT #Wait_Off."Exit" AND #Use.Close AND NOT #FB.Close AND NOT #CMD.Alarm THEN
       #Status := 2;
   END_IF;
   IF #_w1 AND ((#Wait_Off."Exit" AND ((#Use.Close AND NOT #FB.Close) OR (#Use.Open AND #FB.Open))) OR #REQ_OFF.Alarm) THEN
       #Status := 32;
       #Alm.Close := TRUE;
   END_IF;
   IF #_w1 AND #Use.Close AND NOT #FB.Close AND NOT #CMD.Reset THEN #Wait_Off.Start := TRUE; END_IF;
   IF #_w1 THEN #Wait_On.Start := FALSE; END_IF;
   IF #_w1 AND #CMD.Reset THEN #Wait_Off.Start := FALSE; END_IF;
END_REGION

REGION Network 15: Запрос на открытие
   RUNG wire#powerrail
      Contact( #Go )
      I_Contact( #FB.Open )
      I_Contact( #CMD.Sim )
      S_SR(operand := #REQ_Open, r1 := wire#w1)
   END_RUNG
   RUNG wire#powerrail
      I_Contact( #Go )
   END_RUNG wire#w1
   RUNG wire#powerrail
      Contact( #FB.Open )
      Contact( #Use.Electro )
   END_RUNG wire#w1
   RUNG wire#powerrail
      Contact( #CMD.Sim )
   END_RUNG wire#w1
   // the same network as SCL:
   IF #Go AND NOT #FB.Open AND NOT #CMD.Sim THEN
       #REQ_Open := TRUE;   // SR flip-flop
   END_IF;
   IF NOT #Go OR (#FB.Open AND #Use.Electro) OR #CMD.Sim THEN #REQ_Open := FALSE; END_IF;
END_REGION

REGION Network 16: Запрос на закрытие
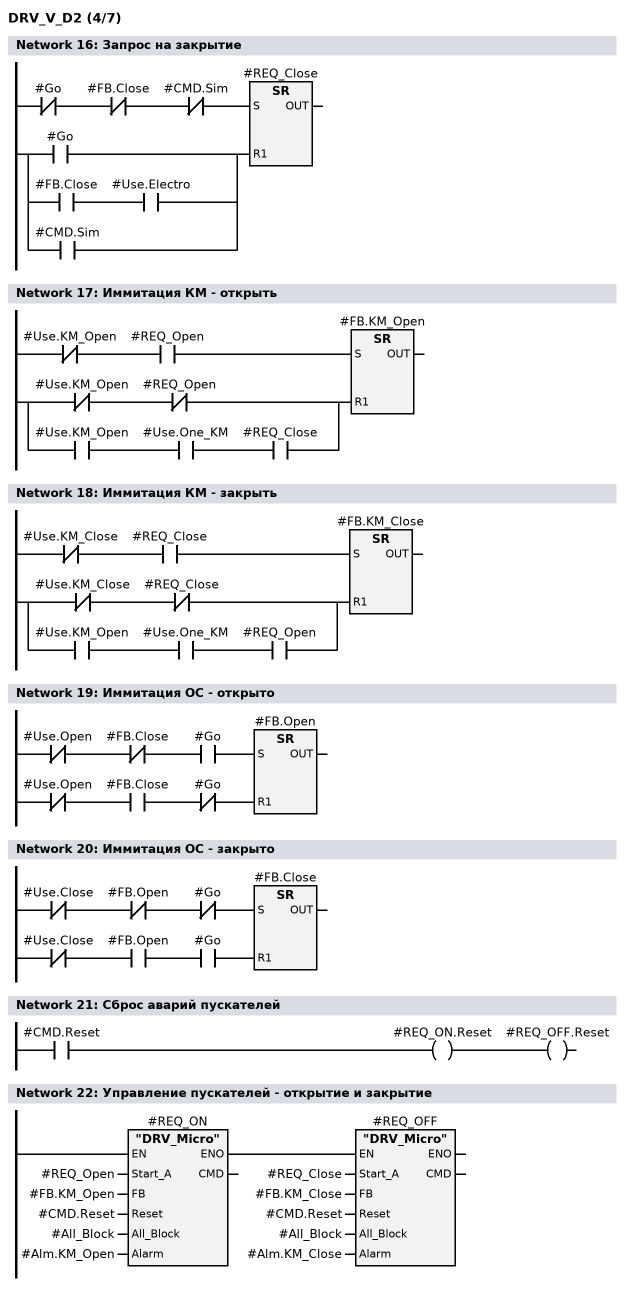
   RUNG wire#powerrail
      I_Contact( #Go )
      I_Contact( #FB.Close )
      I_Contact( #CMD.Sim )
      S_SR(operand := #REQ_Close, r1 := wire#w1)
   END_RUNG
   RUNG wire#powerrail
      Contact( #Go )
   END_RUNG wire#w1
   RUNG wire#powerrail
      Contact( #FB.Close )
      Contact( #Use.Electro )
   END_RUNG wire#w1
   RUNG wire#powerrail
      Contact( #CMD.Sim )
   END_RUNG wire#w1
   // the same network as SCL:
   IF NOT #Go AND NOT #FB.Close AND NOT #CMD.Sim THEN
       #REQ_Close := TRUE;   // SR flip-flop
   END_IF;
   IF #Go OR (#FB.Close AND #Use.Electro) OR #CMD.Sim THEN #REQ_Close := FALSE; END_IF;
END_REGION

REGION Network 17: Иммитация КМ - открыть
   RUNG wire#powerrail
      I_Contact( #Use.KM_Open )
      Contact( #REQ_Open )
      S_SR(operand := #FB.KM_Open, r1 := wire#w1)
   END_RUNG
   RUNG wire#powerrail
      I_Contact( #Use.KM_Open )
      I_Contact( #REQ_Open )
   END_RUNG wire#w1
   RUNG wire#powerrail
      Contact( #Use.KM_Open )
      Contact( #Use.One_KM )
      Contact( #REQ_Close )
   END_RUNG wire#w1
   // the same network as SCL:
   IF NOT #Use.KM_Open AND #REQ_Open THEN
       #FB.KM_Open := TRUE;   // SR flip-flop
   END_IF;
   IF (NOT #Use.KM_Open AND NOT #REQ_Open) OR (#Use.KM_Open AND #Use.One_KM AND #REQ_Close) THEN
       #FB.KM_Open := FALSE;
   END_IF;
END_REGION

REGION Network 18: Иммитация КМ - закрыть
   RUNG wire#powerrail
      I_Contact( #Use.KM_Close )
      Contact( #REQ_Close )
      S_SR(operand := #FB.KM_Close, r1 := wire#w1)
   END_RUNG
   RUNG wire#powerrail
      I_Contact( #Use.KM_Close )
      I_Contact( #REQ_Close )
   END_RUNG wire#w1
   RUNG wire#powerrail
      Contact( #Use.KM_Open )
      Contact( #Use.One_KM )
      Contact( #REQ_Open )
   END_RUNG wire#w1
   // the same network as SCL:
   IF NOT #Use.KM_Close AND #REQ_Close THEN
       #FB.KM_Close := TRUE;   // SR flip-flop
   END_IF;
   IF (NOT #Use.KM_Close AND NOT #REQ_Close) OR (#Use.KM_Open AND #Use.One_KM AND #REQ_Open) THEN
       #FB.KM_Close := FALSE;
   END_IF;
END_REGION

REGION Network 19: Иммитация ОС - открыто
   RUNG wire#powerrail
      I_Contact( #Use.Open )
      I_Contact( #FB.Close )
      Contact( #Go )
      S_SR(operand := #FB.Open, r1 := wire#w1)
   END_RUNG
   RUNG wire#powerrail
      I_Contact( #Use.Open )
      Contact( #FB.Close )
      I_Contact( #Go )
   END_RUNG wire#w1
   // the same network as SCL:
   IF NOT #Use.Open AND NOT #FB.Close AND #Go THEN
       #FB.Open := TRUE;   // SR flip-flop
   END_IF;
   IF NOT #Use.Open AND #FB.Close AND NOT #Go THEN #FB.Open := FALSE; END_IF;
END_REGION

REGION Network 20: Иммитация ОС - закрыто
   RUNG wire#powerrail
      I_Contact( #Use.Close )
      I_Contact( #FB.Open )
      I_Contact( #Go )
      S_SR(operand := #FB.Close, r1 := wire#w1)
   END_RUNG
   RUNG wire#powerrail
      I_Contact( #Use.Close )
      Contact( #FB.Open )
      Contact( #Go )
   END_RUNG wire#w1
   // the same network as SCL:
   IF NOT #Use.Close AND NOT #FB.Open AND NOT #Go THEN
       #FB.Close := TRUE;   // SR flip-flop
   END_IF;
   IF NOT #Use.Close AND #FB.Open AND #Go THEN #FB.Close := FALSE; END_IF;
END_REGION

REGION Network 21: Сброс аварий пускателей
   RUNG wire#powerrail
      Contact( #CMD.Reset )
      Coil( #REQ_ON.Reset )
      Coil( #REQ_OFF.Reset )
   END_RUNG
   // the same network as SCL:
   #REQ_ON.Reset := #CMD.Reset;
   #REQ_OFF.Reset := #CMD.Reset;
END_REGION

REGION Network 22: Управление пускателей - открытие и закрытие
   RUNG wire#powerrail
      #REQ_ON(Start_A := #REQ_Open, FB := #FB.KM_Open, Reset := #CMD.Reset, All_Block := #All_Block, Alarm := #Alm.KM_Open, CMD =>)
      #REQ_OFF(Start_A := #REQ_Close, FB := #FB.KM_Close, Reset := #CMD.Reset, All_Block := #All_Block, Alarm := #Alm.KM_Close, CMD =>)
   END_RUNG
   // the same network as SCL:
   #REQ_ON(Start_A := #REQ_Open,   // "DRV_Micro"
           FB := #FB.KM_Open,
           Reset := #CMD.Reset,
           All_Block := #All_Block,
           Alarm := #Alm.KM_Open,
           ENO => #_w1);
   IF #_w1 THEN
       #REQ_OFF(Start_A := #REQ_Close,   // "DRV_Micro"
                FB := #FB.KM_Close,
                Reset := #CMD.Reset,
                All_Block := #All_Block,
                Alarm := #Alm.KM_Close);
   END_IF;
END_REGION

REGION Network 23: Команда - открыть
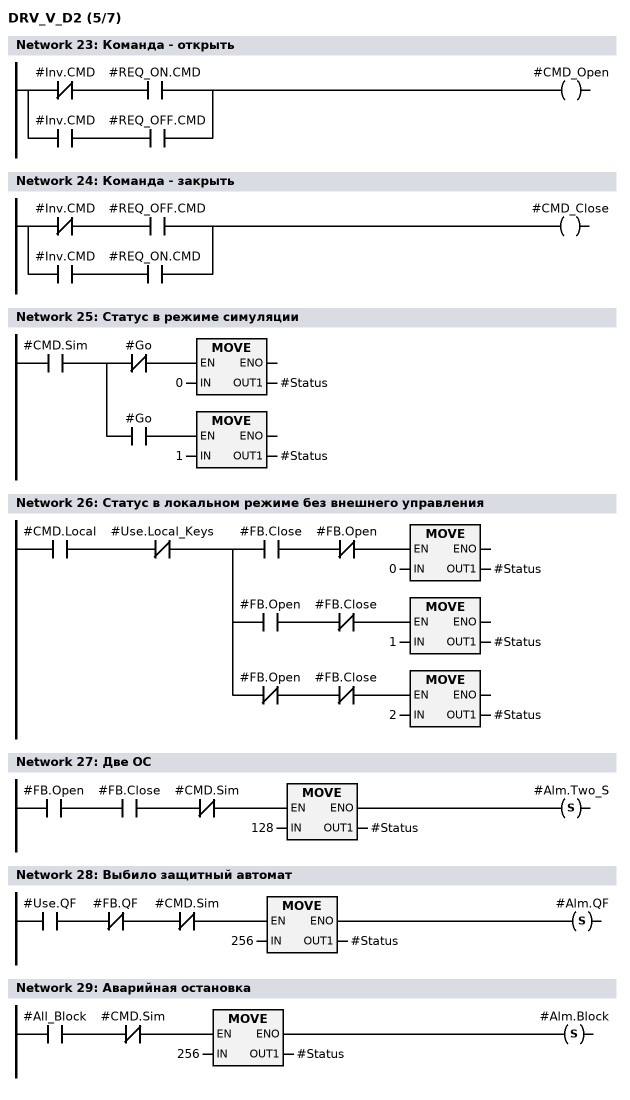
   RUNG wire#powerrail
      I_Contact( #Inv.CMD )
      Contact( #REQ_ON.CMD )
      wire#w1
      Coil( #CMD_Open )
   END_RUNG
   RUNG wire#powerrail
      Contact( #Inv.CMD )
      Contact( #REQ_OFF.CMD )
   END_RUNG wire#w1
   // the same network as SCL:
   #CMD_Open := (NOT #Inv.CMD AND #REQ_ON.CMD) OR (#Inv.CMD AND #REQ_OFF.CMD);
END_REGION

REGION Network 24: Команда - закрыть
   RUNG wire#powerrail
      I_Contact( #Inv.CMD )
      Contact( #REQ_OFF.CMD )
      wire#w1
      Coil( #CMD_Close )
   END_RUNG
   RUNG wire#powerrail
      Contact( #Inv.CMD )
      Contact( #REQ_ON.CMD )
   END_RUNG wire#w1
   // the same network as SCL:
   #CMD_Close := (NOT #Inv.CMD AND #REQ_OFF.CMD) OR (#Inv.CMD AND #REQ_ON.CMD);
END_REGION

REGION Network 25: Статус в режиме симуляции
   RUNG wire#powerrail
      Contact( #CMD.Sim )
      wire#w1
      I_Contact( #Go )
      Move(in := 0, out1 => #Status)
   END_RUNG
   RUNG wire#w1
      Contact( #Go )
      Move(in := 1, out1 => #Status)
   END_RUNG
   // the same network as SCL:
   IF #CMD.Sim AND NOT #Go THEN #Status := 0; END_IF;
   IF #CMD.Sim AND #Go THEN #Status := 1; END_IF;
END_REGION

REGION Network 26: Статус в локальном режиме без внешнего управления
   RUNG wire#powerrail
      Contact( #CMD.Local )
      I_Contact( #Use.Local_Keys )
      wire#w1
      Contact( #FB.Close )
      I_Contact( #FB.Open )
      Move(in := 0, out1 => #Status)
   END_RUNG
   RUNG wire#w1
      Contact( #FB.Open )
      I_Contact( #FB.Close )
      Move(in := 1, out1 => #Status)
   END_RUNG
   RUNG wire#w1
      I_Contact( #FB.Open )
      I_Contact( #FB.Close )
      Move(in := 2, out1 => #Status)
   END_RUNG
   // the same network as SCL:
   #_w1 := #CMD.Local AND NOT #Use.Local_Keys;
   IF #_w1 AND #FB.Close AND NOT #FB.Open THEN #Status := 0; END_IF;
   IF #_w1 AND #FB.Open AND NOT #FB.Close THEN #Status := 1; END_IF;
   IF #_w1 AND NOT #FB.Open AND NOT #FB.Close THEN #Status := 2; END_IF;
END_REGION

REGION Network 27: Две ОС
   RUNG wire#powerrail
      Contact( #FB.Open )
      Contact( #FB.Close )
      I_Contact( #CMD.Sim )
      Move(in := 128, out1 => #Status)
      S_Coil( #Alm.Two_S )
   END_RUNG
   // the same network as SCL:
   IF #FB.Open AND #FB.Close AND NOT #CMD.Sim THEN
       #Status := 128;
       #Alm.Two_S := TRUE;
   END_IF;
END_REGION

REGION Network 28: Выбило защитный автомат
   RUNG wire#powerrail
      Contact( #Use.QF )
      I_Contact( #FB.QF )
      I_Contact( #CMD.Sim )
      Move(in := 256, out1 => #Status)
      S_Coil( #Alm.QF )
   END_RUNG
   // the same network as SCL:
   IF #Use.QF AND NOT #FB.QF AND NOT #CMD.Sim THEN
       #Status := 256;
       #Alm.QF := TRUE;
   END_IF;
END_REGION

REGION Network 29: Аварийная остановка
   RUNG wire#powerrail
      Contact( #All_Block )
      I_Contact( #CMD.Sim )
      Move(in := 256, out1 => #Status)
      S_Coil( #Alm.Block )
   END_RUNG
   // the same network as SCL:
   IF #All_Block AND NOT #CMD.Sim THEN
       #Status := 256;
       #Alm.Block := TRUE;
   END_IF;
END_REGION

REGION Network 30: Авария
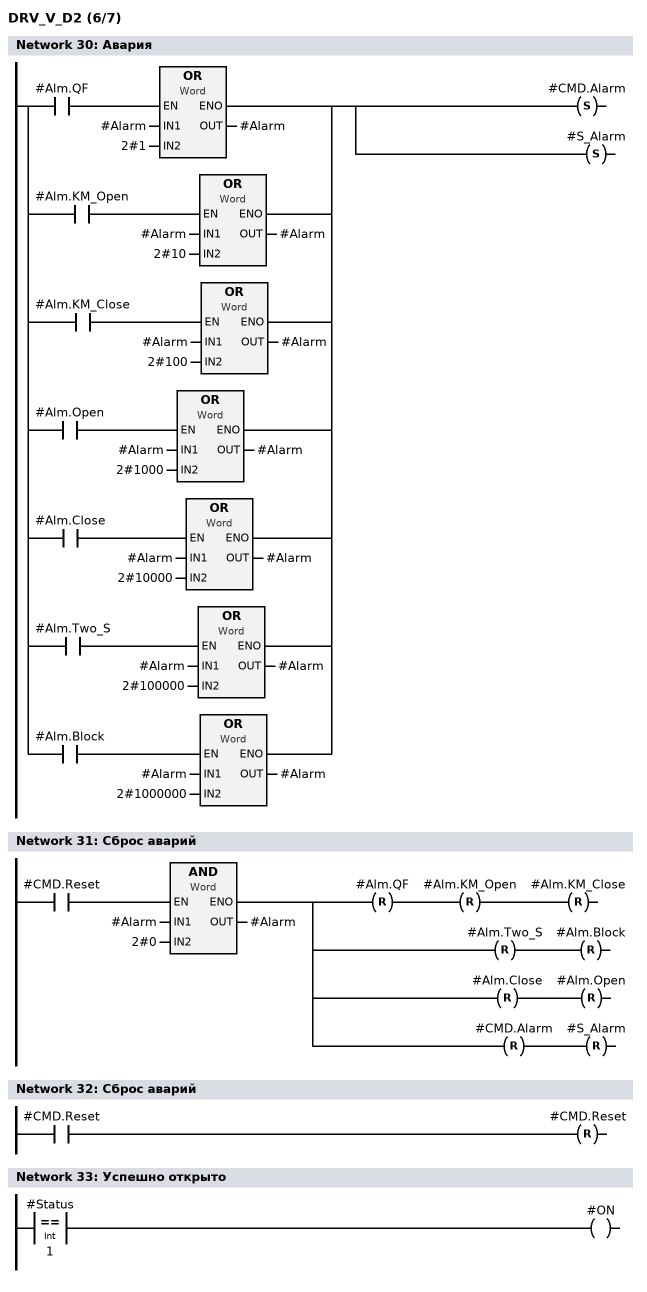
   // no checked SCL form for this network; see the picture
END_REGION

REGION Network 31: Сброс аварий
   // no checked SCL form for this network; see the picture
END_REGION

REGION Network 32: Сброс аварий
   RUNG wire#powerrail
      Contact( #CMD.Reset )
      R_Coil( #CMD.Reset )
   END_RUNG
   // the same network as SCL:
   IF #CMD.Reset THEN #CMD.Reset := FALSE; END_IF;
END_REGION

REGION Network 33: Успешно открыто
   RUNG wire#powerrail
      { S7_Templates := "SrcType := Int" } EQ_Contact(in1 := #Status, in2 := 1)
      Coil( #ON )
   END_RUNG
   // the same network as SCL:
   #ON := #Status = 1;
END_REGION

REGION Network 34: Успешно закрыто
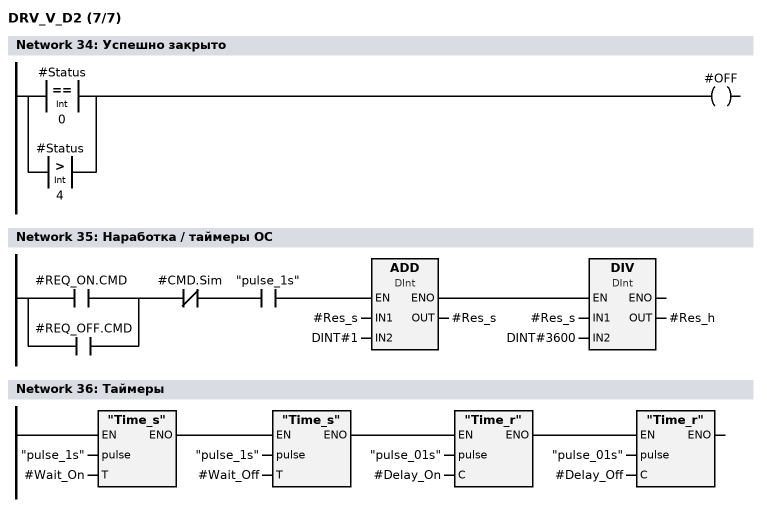
   RUNG wire#powerrail
      { S7_Templates := "SrcType := Int" } EQ_Contact(in1 := #Status, in2 := 0)
      wire#w1
      Coil( #OFF )
   END_RUNG
   RUNG wire#powerrail
      { S7_Templates := "SrcType := Int" } GT_Contact(in1 := #Status, in2 := 4)
   END_RUNG wire#w1
   // the same network as SCL:
   #OFF := (#Status = 0) OR (#Status > 4);
END_REGION

REGION Network 35: Наработка / таймеры ОС
   RUNG wire#powerrail
      Contact( #REQ_ON.CMD )
      wire#w1
      I_Contact( #CMD.Sim )
      Contact( "pulse_1s" )
      { S7_Templates := "SrcType := DInt"; S7_GenerateENO := "TRUE" } Add(in1 := #Res_s, in2 := DINT#1, out => #Res_s)
      { S7_Templates := "SrcType := DInt"; S7_GenerateENO := "TRUE" } Div(in1 := #Res_s, in2 := DINT#3600, out => #Res_h)
   END_RUNG
   RUNG wire#powerrail
      Contact( #REQ_OFF.CMD )
   END_RUNG wire#w1
   // the same network as SCL:
   // ENO of a box is taken as its EN; it also drops when the box reports an error
   IF (#REQ_ON.CMD OR #REQ_OFF.CMD) AND NOT #CMD.Sim AND "pulse_1s" THEN
       #Res_s := #Res_s + DINT#1;
       #Res_h := #Res_s / DINT#3600;
   END_IF;
END_REGION

REGION Network 36: Таймеры
   RUNG wire#powerrail
      "Time_s"(pulse := "pulse_1s", T := #Wait_On)
      "Time_s"(pulse := "pulse_1s", T := #Wait_Off)
      "Time_r"(pulse := "pulse_01s", C := #Delay_On)
      "Time_r"(pulse := "pulse_01s", C := #Delay_Off)
   END_RUNG
   // the same network as SCL:
   "Time_s"(pulse := "pulse_1s", T := #Wait_On, ENO => #_w1);
   "Time_s"(EN := #_w1, pulse := "pulse_1s", T := #Wait_Off, ENO => #_w2);
   "Time_r"(EN := #_w2, pulse := "pulse_01s", C := #Delay_On, ENO => #_w3);
   IF #_w3 THEN "Time_r"(pulse := "pulse_01s", C := #Delay_Off); END_IF;
END_REGION
END_FUNCTION_BLOCK

// folder: DRV_Low

FUNCTION_BLOCK "DI_ex"   // FB100, LAD
{ S7_Optimized_Access := 'FALSE' }
VERSION : 0.1
   VAR_INPUT
      Input : Bool;   // Входящий сигнал
      pulse : Bool;   // Частота фильтрации дребезка
   END_VAR
   VAR_OUTPUT
      Signal : Bool;   // Результирующий сигнал
   END_VAR
   VAR
      Hand : Bool;   // 0 - Авто, 1 - Ручной
      Start_M : Bool;   // Запуск в ручном режиме
      Data : Bool;   // Отфильтрованный сигнал
      Inverse : Bool;   // Инверсия входного сигнала
      Filter_On : Struct   // Фильтр наличия сигнала
         SP : Int;
         Now : Int;
         "Exit" : Bool;
         Start : Bool;
         Pause : Bool;
         Reset : Bool;
      END_STRUCT;
      Filter_Off : Struct   // Фильтр отсутствия сигнала
         SP : Int;
         Now : Int;
         "Exit" : Bool;
         Start : Bool;
         Pause : Bool;
         Reset : Bool;
      END_STRUCT;
      res_1 : Word;
   END_VAR
   VAR_TEMP   // added for the SCL form of the ladder/FBD networks
      _w1 : Bool;
   END_VAR
BEGIN

REGION Network 1: Устройство в ручном режиме
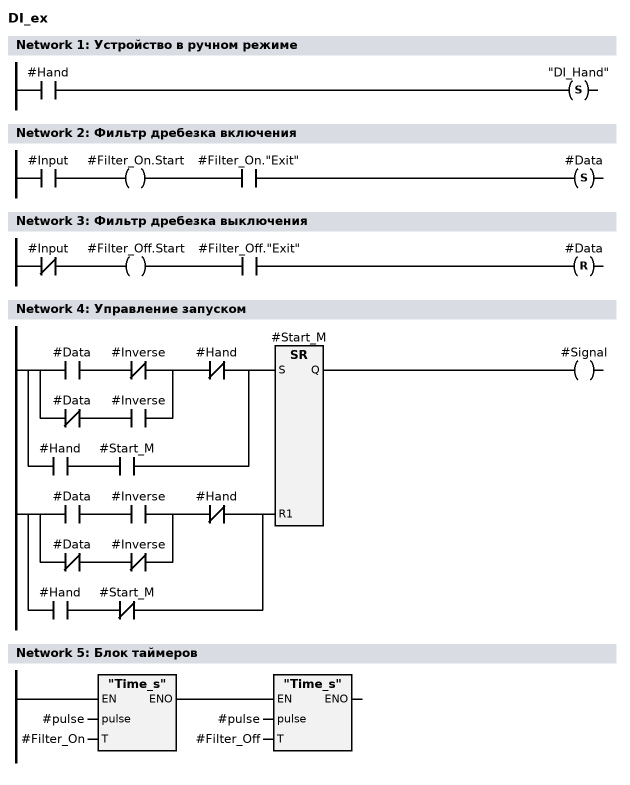
   RUNG wire#powerrail
      Contact( #Hand )
      S_Coil( "DI_Hand" )
   END_RUNG
   // the same network as SCL:
   IF #Hand THEN "DI_Hand" := TRUE; END_IF;
END_REGION

REGION Network 2: Фильтр дребезка включения
   RUNG wire#powerrail
      Contact( #Input )
      Coil( #Filter_On.Start )
      Contact( #Filter_On."Exit" )
      S_Coil( #Data )
   END_RUNG
   // the same network as SCL:
   #Filter_On.Start := #Input;
   IF #Input AND #Filter_On."Exit" THEN #Data := TRUE; END_IF;
END_REGION

REGION Network 3: Фильтр дребезка выключения
   RUNG wire#powerrail
      I_Contact( #Input )
      Coil( #Filter_Off.Start )
      Contact( #Filter_Off."Exit" )
      R_Coil( #Data )
   END_RUNG
   // the same network as SCL:
   #Filter_Off.Start := NOT #Input;
   IF NOT #Input AND #Filter_Off."Exit" THEN #Data := FALSE; END_IF;
END_REGION

REGION Network 4: Управление запуском
   RUNG wire#powerrail
      Contact( #Data )
      I_Contact( #Inverse )
      wire#w1
      I_Contact( #Hand )
      wire#w2
      S_SR(operand := #Start_M, r1 := wire#w4)
      Coil( #Signal )
   END_RUNG
   RUNG wire#powerrail
      I_Contact( #Data )
      Contact( #Inverse )
   END_RUNG wire#w1
   RUNG wire#powerrail
      Contact( #Hand )
      Contact( #Start_M )
   END_RUNG wire#w2
   RUNG wire#powerrail
      Contact( #Data )
      Contact( #Inverse )
      wire#w3
      I_Contact( #Hand )
   END_RUNG wire#w4
   RUNG wire#powerrail
      I_Contact( #Data )
      I_Contact( #Inverse )
   END_RUNG wire#w3
   RUNG wire#powerrail
      Contact( #Hand )
      I_Contact( #Start_M )
   END_RUNG wire#w4
   // the same network as SCL:
   #_w1 := (((#Data AND #Inverse) OR (NOT #Data AND NOT #Inverse)) AND NOT #Hand) OR (#Hand AND NOT #Start_M);
   IF (((#Data AND NOT #Inverse) OR (NOT #Data AND #Inverse)) AND NOT #Hand) OR (#Hand AND #Start_M) THEN
       #Start_M := TRUE;   // SR flip-flop
   END_IF;
   IF #_w1 THEN #Start_M := FALSE; END_IF;
   #Signal := #Start_M;
END_REGION

REGION Network 5: Блок таймеров
   RUNG wire#powerrail
      "Time_s"(pulse := #pulse, T := #Filter_On)
      "Time_s"(pulse := #pulse, T := #Filter_Off)
   END_RUNG
   // the same network as SCL:
   "Time_s"(pulse := #pulse, T := #Filter_On, ENO => #_w1);
   IF #_w1 THEN "Time_s"(pulse := #pulse, T := #Filter_Off); END_IF;
END_REGION
END_FUNCTION_BLOCK

FUNCTION_BLOCK "DO_ex"   // FB101, LAD
{ S7_Optimized_Access := 'FALSE' }
VERSION : 0.1
   VAR_IN_OUT
      Start : Bool;   // Управляющий сигнал из программы
      pulse : Bool;   // Частота длительности импульса
      Q : Bool;   // Выходной сигнал контроллера
   END_VAR
   VAR
      Hand : Bool;   // 0 - Авто, 1 - Ручной
      Start_M : Bool;   // Запуск в ручном режиме
      Simulation : Bool;   // Режим симуляции
      Inverse : Bool;   // Инверсия выхода
      Impulse : Bool;   // Импульсный режим
      T_Impulse : Struct   // Длительность импульса
         SP : Int := 5;
         Now : Int;
         "Exit" : Bool;
         Start : Bool;
         Pause : Bool;
         Reset : Bool;
      END_STRUCT;
   END_VAR
   VAR_TEMP   // added for the SCL form of the ladder/FBD networks
      _w1 : Bool;
   END_VAR
BEGIN

REGION Network 1: Устройство в ручном режиме
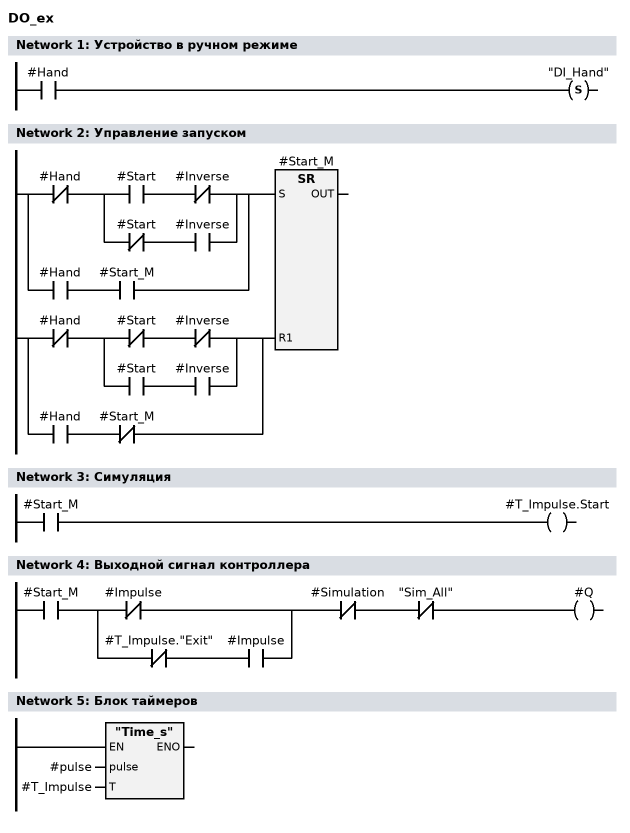
   RUNG wire#powerrail
      Contact( #Hand )
      S_Coil( "DI_Hand" )
   END_RUNG
   // the same network as SCL:
   IF #Hand THEN "DI_Hand" := TRUE; END_IF;
END_REGION

REGION Network 2: Управление запуском
   RUNG wire#powerrail
      I_Contact( #Hand )
      wire#w1
      Contact( #Start )
      I_Contact( #Inverse )
      wire#w2
      S_SR(operand := #Start_M, r1 := wire#w4)
   END_RUNG
   RUNG wire#w1
      I_Contact( #Start )
      Contact( #Inverse )
   END_RUNG wire#w2
   RUNG wire#powerrail
      Contact( #Hand )
      Contact( #Start_M )
   END_RUNG wire#w2
   RUNG wire#powerrail
      I_Contact( #Hand )
      wire#w3
      I_Contact( #Start )
      I_Contact( #Inverse )
   END_RUNG wire#w4
   RUNG wire#w3
      Contact( #Start )
      Contact( #Inverse )
   END_RUNG wire#w4
   RUNG wire#powerrail
      Contact( #Hand )
      I_Contact( #Start_M )
   END_RUNG wire#w4
   // the same network as SCL:
   #_w1 := (NOT #Hand AND ((NOT #Start AND NOT #Inverse) OR (#Start AND #Inverse))) OR (#Hand AND NOT #Start_M);
   IF (NOT #Hand AND ((#Start AND NOT #Inverse) OR (NOT #Start AND #Inverse))) OR (#Hand AND #Start_M) THEN
       #Start_M := TRUE;   // SR flip-flop
   END_IF;
   IF #_w1 THEN #Start_M := FALSE; END_IF;
END_REGION

REGION Network 3: Симуляция
   RUNG wire#powerrail
      Contact( #Start_M )
      Coil( #T_Impulse.Start )
   END_RUNG
   // the same network as SCL:
   #T_Impulse.Start := #Start_M;
END_REGION

REGION Network 4: Выходной сигнал контроллера
   RUNG wire#powerrail
      Contact( #Start_M )
      wire#w1
      I_Contact( #Impulse )
      wire#w2
      I_Contact( #Simulation )
      I_Contact( "Sim_All" )
      Coil( #Q )
   END_RUNG
   RUNG wire#w1
      I_Contact( #T_Impulse."Exit" )
      Contact( #Impulse )
   END_RUNG wire#w2
   // the same network as SCL:
   #Q := #Start_M AND (NOT #Impulse OR (NOT #T_Impulse."Exit" AND #Impulse)) AND NOT #Simulation AND NOT "Sim_All";
END_REGION

REGION Network 5: Блок таймеров
   RUNG wire#powerrail
      "Time_s"(pulse := #pulse, T := #T_Impulse)
   END_RUNG
   // the same network as SCL:
   "Time_s"(pulse := #pulse, T := #T_Impulse);
END_REGION
END_FUNCTION_BLOCK

FUNCTION_BLOCK "AI_ex"   // FB102, LAD
{ S7_Optimized_Access := 'FALSE' }
VERSION : 0.1
   VAR_INPUT
      Signal : Int;   // Входной сигнал контроллера
      All_Block : Bool;   // Аварийная остановка
      pulse : Bool;   // Частота фильтрации сигнала
   END_VAR
   VAR_IN_OUT
      S_Alarm : Bool;   // Наличие аварии
      Result : Real;   // Результат измерений
   END_VAR
   VAR
      CMD : Struct   // Основные команды / Блок команд
         Hand : Bool;   // 0 - авто, 1 - ручной / 0 - Авто, 1 - Ручной
         Start_A : Bool := True;   // Автозапуск / Запуск в авторежиме
         Start_M : Bool;   // Ручной - вперёд / Запуск в ручном режиме
         Force : Bool;   // Принудительный
         Lock : Bool;   // Блокировать / Блокировка
         Local : Bool;   // Локальный
         Service : Bool;   // Сервис
         Safety : Bool;   // Безопасность
         Alarm : Bool;   // Есть авария / Авария
         Reset : Bool;   // Сброс аварий
         Sim : Bool;   // Режим симуляции
      END_STRUCT;
      Mode : Int;   // Режим работы
      Status : Int;   // Статус устройства
      Use : Struct   // Функционал
         RTD : Bool;   // Режим RTD
         Filter : Bool;   // Филтрация сигнала
         Inverse : Bool;   // Инверсия сигнала
      END_STRUCT;
      Signal_DI : DInt;   // Конвертация сигнала
      Signal_R : Real;   // Конвертация сигнала
      Value : Real;   // Итоговый сигнал
      RTD_c : Real := 10.0;   // Коэффициент RTD
      Calibration : Real;   // Поправка
      Filter : Struct   // Фильтрация сигнала
         SP : Real := 5.0;
         Now : Real;
         Summ : Real;
         Result : Real;
         Last : Real;
      END_STRUCT;
      Converter : Struct   // Масштабирование сигнала
         Use_Min_In : Bool;   // Отсекать входные значения ниже минимума
         Use_Max_In : Bool;   // Отсекать входные значения выше максимума
         Use_Min_Out : Bool;   // Отсекать результат ниже минимума
         Use_Max_Out : Bool;   // Отсекать результат выше максимума
         IO : Bool;   // Входной/Выходной режим
         Inverse : Bool;   // Инверсия выхода
         Min_In : Real;   // Минимальный входной сигнал
         Max_In : Real := 27648.0;   // Максимальный входной сигнал
         Min_Out : Real;   // Минимальный выходной сигнал
         Max_Out : Real := 100.0;   // Максимальный выходной сигнал
      END_STRUCT;
      SP : Struct   // Уставки аварий
         NC : Real := -500.0;
         SC : Real := 28000.0;
         HH : Real := 90.0;
         H : Real := 85.0;
         L : Real := 15.0;
         LL : Real := 10.0;
      END_STRUCT;
      Timers : Struct   // Таймеры аварий
         NC : Struct
            SP : Int := 10;
            Now : Int;
            "Exit" : Bool;
            Start : Bool;
            Pause : Bool;
            Reset : Bool;
         END_STRUCT;
         SC : Struct
            SP : Int := 10;
            Now : Int;
            "Exit" : Bool;
            Start : Bool;
            Pause : Bool;
            Reset : Bool;
         END_STRUCT;
         HH : Struct
            SP : Int;
            Now : Int;
            "Exit" : Bool;
            Start : Bool;
            Pause : Bool;
            Reset : Bool;
         END_STRUCT;
         H : Struct
            SP : Int := 5;
            Now : Int;
            "Exit" : Bool;
            Start : Bool;
            Pause : Bool;
            Reset : Bool;
         END_STRUCT;
         L : Struct
            SP : Int := 5;
            Now : Int;
            "Exit" : Bool;
            Start : Bool;
            Pause : Bool;
            Reset : Bool;
         END_STRUCT;
         LL : Struct
            SP : Int;
            Now : Int;
            "Exit" : Bool;
            Start : Bool;
            Pause : Bool;
            Reset : Bool;
         END_STRUCT;
      END_STRUCT;
      Alarms : Struct   // Список аварий
         NC : Bool;   // обрыв линии
         SC : Bool;   // короткое замыкание
         HH : Bool;
         H : Bool;
         L : Bool;
         LL : Bool;
      END_STRUCT;
      Alarm : Word;   // Слово аварий
   END_VAR
   VAR_TEMP   // added for the SCL form of the ladder/FBD networks
      _w1 : Bool;
      _w2 : Bool;
   END_VAR
BEGIN

REGION Network 1: Общий сброс
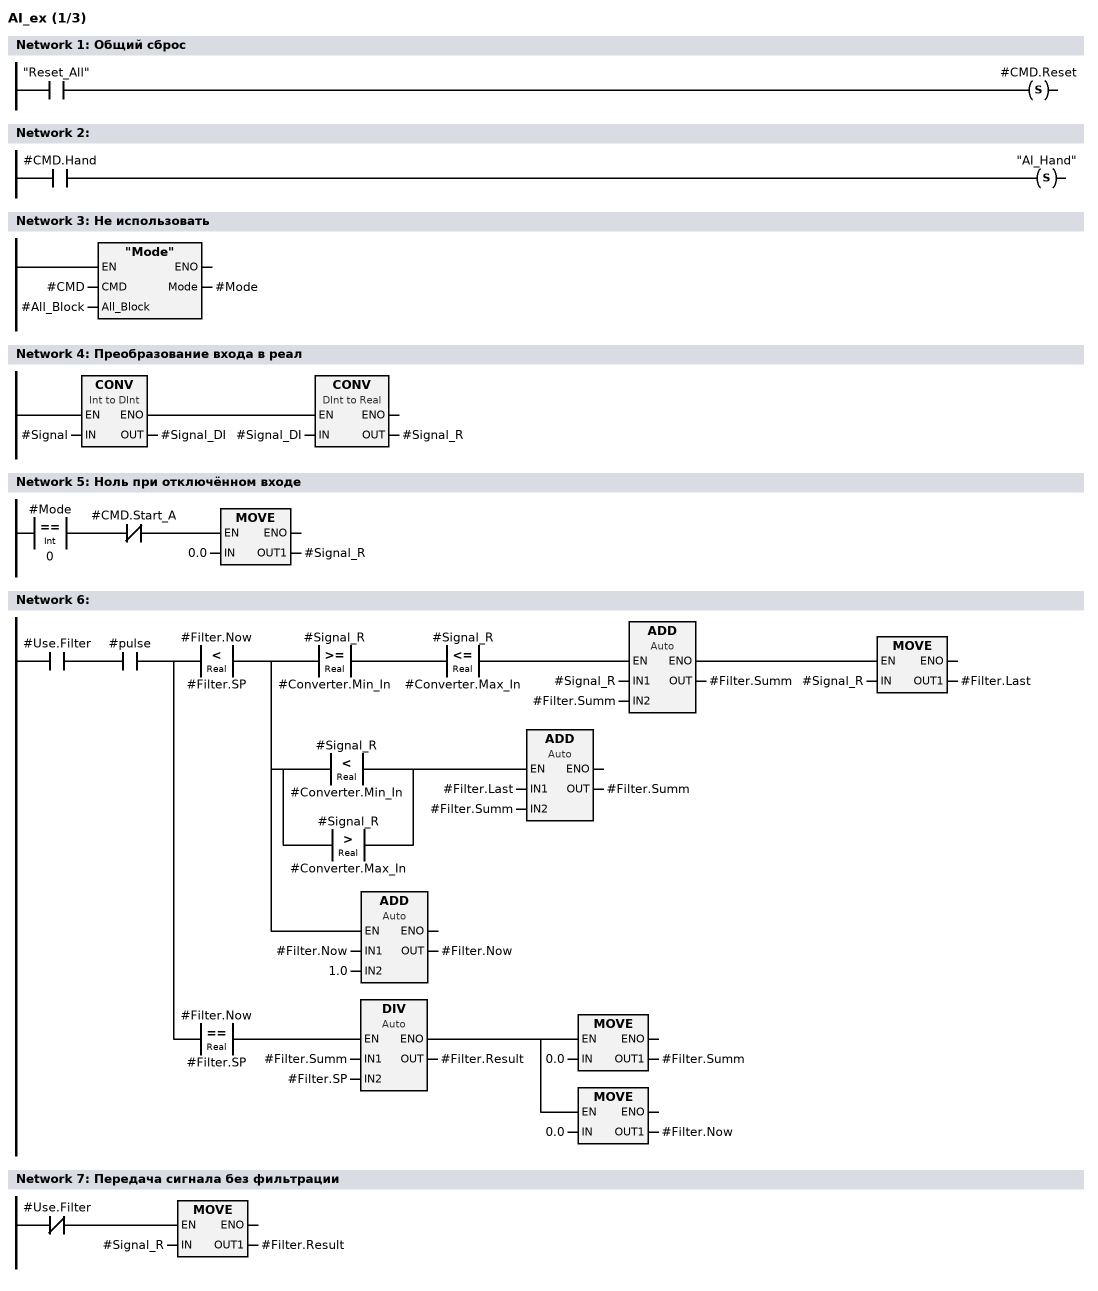
   RUNG wire#powerrail
      Contact( "Reset_All" )
      S_Coil( #CMD.Reset )
   END_RUNG
   // the same network as SCL:
   IF "Reset_All" THEN #CMD.Reset := TRUE; END_IF;
END_REGION

REGION Network 2
   RUNG wire#powerrail
      Contact( #CMD.Hand )
      S_Coil( "AI_Hand" )
   END_RUNG
   // the same network as SCL:
   IF #CMD.Hand THEN "AI_Hand" := TRUE; END_IF;
END_REGION

REGION Network 3: Не использовать
   RUNG wire#powerrail
      "Mode"(CMD := #CMD, All_Block := #All_Block, Mode => #Mode)
   END_RUNG
   // the same network as SCL:
   "Mode"(CMD := #CMD, All_Block := #All_Block, Mode => #Mode);
END_REGION

REGION Network 4: Преобразование входа в реал
   RUNG wire#powerrail
      { S7_Templates := "[SrcType := Int, DestType := DInt]"; S7_GenerateENO := "TRUE" } Convert(in := #Signal, out => #Signal_DI)
      { S7_Templates := "[SrcType := DInt, DestType := Real]"; S7_GenerateENO := "TRUE" } Convert(in := #Signal_DI, out => #Signal_R)
   END_RUNG
   // the same network as SCL:
   // ENO of a box is taken as its EN; it also drops when the box reports an error
   #Signal_DI := INT_TO_DINT(#Signal);
   #Signal_R := DINT_TO_REAL(#Signal_DI);
END_REGION

REGION Network 5: Ноль при отключённом входе
   RUNG wire#powerrail
      { S7_Templates := "SrcType := Int" } EQ_Contact(in1 := #Mode, in2 := 0)
      I_Contact( #CMD.Start_A )
      Move(in := 0.0, out1 => #Signal_R)
   END_RUNG
   // the same network as SCL:
   IF (#Mode = 0) AND NOT #CMD.Start_A THEN #Signal_R := 0.0; END_IF;
END_REGION

REGION Network 6
   RUNG wire#powerrail
      Contact( #Use.Filter )
      Contact( #pulse )
      wire#w1
      { S7_Templates := "SrcType := Real" } LT_Contact(in1 := #Filter.Now, in2 := #Filter.SP)
      wire#w2
      { S7_Templates := "SrcType := Real" } GE_Contact(in1 := #Signal_R, in2 := #Converter.Min_In)
      { S7_Templates := "SrcType := Real" } LE_Contact(in1 := #Signal_R, in2 := #Converter.Max_In)
      Add(in1 := #Signal_R, in2 := #Filter.Summ, out => #Filter.Summ)
      Move(in := #Signal_R, out1 => #Filter.Last)
   END_RUNG
   RUNG wire#w2
      { S7_Templates := "SrcType := Real" } LT_Contact(in1 := #Signal_R, in2 := #Converter.Min_In)
      wire#w3
      Add(in1 := #Filter.Last, in2 := #Filter.Summ, out => #Filter.Summ)
   END_RUNG
   RUNG wire#w2
      { S7_Templates := "SrcType := Real" } GT_Contact(in1 := #Signal_R, in2 := #Converter.Max_In)
   END_RUNG wire#w3
   RUNG wire#w2
      Add(in1 := #Filter.Now, in2 := 1.0, out => #Filter.Now)
   END_RUNG
   RUNG wire#w1
      { S7_Templates := "SrcType := Real" } EQ_Contact(in1 := #Filter.Now, in2 := #Filter.SP)
      Div(in1 := #Filter.Summ, in2 := #Filter.SP, out => #Filter.Result)
      wire#w4
      Move(in := 0.0, out1 => #Filter.Summ)
   END_RUNG
   RUNG wire#w4
      Move(in := 0.0, out1 => #Filter.Now)
   END_RUNG
   // the same network as SCL:
   #_w1 := #Use.Filter AND #pulse;
   #_w2 := #_w1 AND (#Filter.Now < #Filter.SP);
   IF #_w2 AND (#Signal_R >= #Converter.Min_In) AND (#Signal_R <= #Converter.Max_In) THEN
       #Filter.Summ := #Signal_R + #Filter.Summ;
       #Filter.Last := #Signal_R;
   END_IF;
   IF #_w2 AND ((#Signal_R < #Converter.Min_In) OR (#Signal_R > #Converter.Max_In)) THEN
       #Filter.Summ := #Filter.Last + #Filter.Summ;
   END_IF;
   IF #_w2 THEN #Filter.Now := #Filter.Now + 1.0; END_IF;
   IF #_w1 AND (#Filter.Now = #Filter.SP) THEN
       #Filter.Result := #Filter.Summ / #Filter.SP;
       #Filter.Summ := 0.0;
       #Filter.Now := 0.0;
   END_IF;
END_REGION

REGION Network 7: Передача сигнала без фильтрации
   RUNG wire#powerrail
      I_Contact( #Use.Filter )
      { S7_GenerateENO := "TRUE" } Move(in := #Signal_R, out1 => #Filter.Result)
   END_RUNG
   // the same network as SCL:
   IF NOT #Use.Filter THEN #Filter.Result := #Signal_R; END_IF;
END_REGION

REGION Network 8: Режим РТД
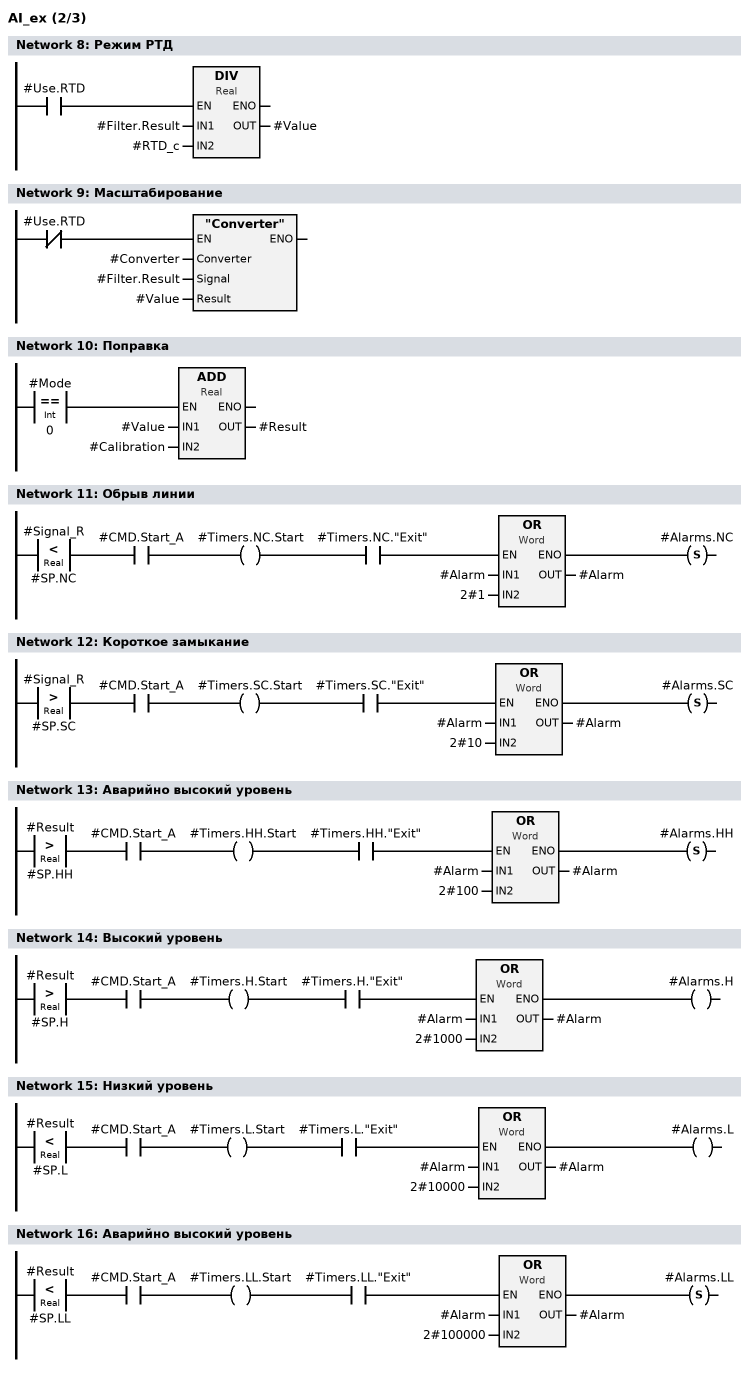
   RUNG wire#powerrail
      Contact( #Use.RTD )
      { S7_Templates := "SrcType := Real"; S7_GenerateENO := "TRUE" } Div(in1 := #Filter.Result, in2 := #RTD_c, out => #Value)
   END_RUNG
   // the same network as SCL:
   IF #Use.RTD THEN #Value := #Filter.Result / #RTD_c; END_IF;
END_REGION

REGION Network 9: Масштабирование
   RUNG wire#powerrail
      I_Contact( #Use.RTD )
      "Converter"(Converter := #Converter, Signal := #Filter.Result, Result := #Value)
   END_RUNG
   // the same network as SCL:
   IF NOT #Use.RTD THEN
       "Converter"(Converter := #Converter, Signal := #Filter.Result, Result := #Value);
   END_IF;
END_REGION

REGION Network 10: Поправка
   RUNG wire#powerrail
      { S7_Templates := "SrcType := Int" } EQ_Contact(in1 := #Mode, in2 := 0)
      { S7_Templates := "SrcType := Real"; S7_GenerateENO := "TRUE" } Add(in1 := #Value, in2 := #Calibration, out => #Result)
   END_RUNG
   // the same network as SCL:
   IF #Mode = 0 THEN #Result := #Value + #Calibration; END_IF;
END_REGION

REGION Network 11: Обрыв линии
   // no checked SCL form for this network; see the picture
END_REGION

REGION Network 12: Короткое замыкание
   // no checked SCL form for this network; see the picture
END_REGION

REGION Network 13: Аварийно высокий уровень
   // no checked SCL form for this network; see the picture
END_REGION

REGION Network 14: Высокий уровень
   // no checked SCL form for this network; see the picture
END_REGION

REGION Network 15: Низкий уровень
   // no checked SCL form for this network; see the picture
END_REGION

REGION Network 16: Аварийно высокий уровень
   // no checked SCL form for this network; see the picture
END_REGION

REGION Network 17: Наличие любой ошибки
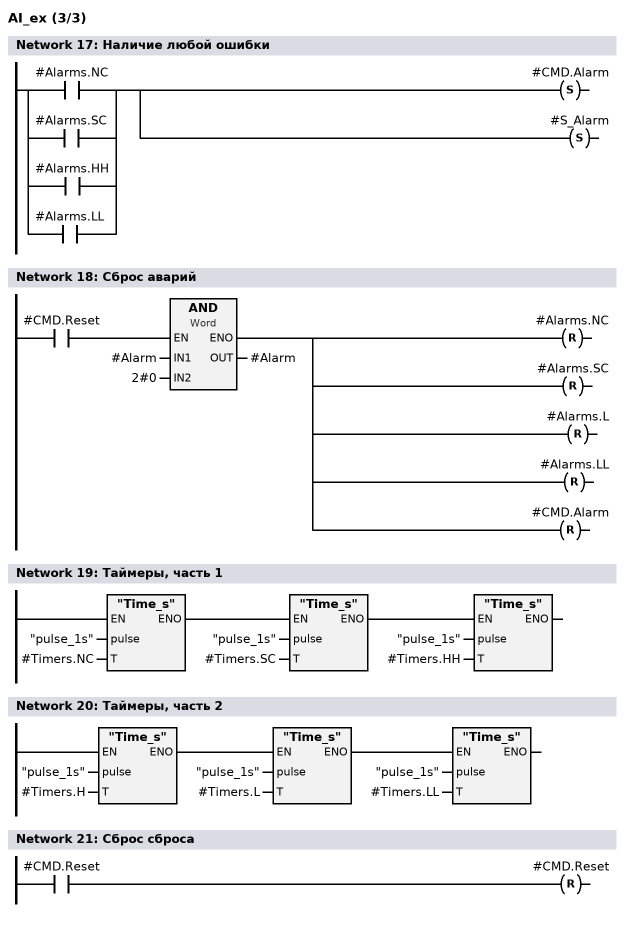
   RUNG wire#powerrail
      Contact( #Alarms.NC )
      wire#w1
      S_Coil( #CMD.Alarm )
   END_RUNG
   RUNG wire#powerrail
      Contact( #Alarms.SC )
   END_RUNG wire#w1
   RUNG wire#powerrail
      Contact( #Alarms.HH )
   END_RUNG wire#w1
   RUNG wire#powerrail
      Contact( #Alarms.LL )
   END_RUNG wire#w1
   RUNG wire#w1
      S_Coil( #S_Alarm )
   END_RUNG
   // the same network as SCL:
   IF #Alarms.NC OR #Alarms.SC OR #Alarms.HH OR #Alarms.LL THEN
       #CMD.Alarm := TRUE;
       #S_Alarm := TRUE;
   END_IF;
END_REGION

REGION Network 18: Сброс аварий
   // no checked SCL form for this network; see the picture
END_REGION

REGION Network 19: Таймеры, часть 1
   RUNG wire#powerrail
      "Time_s"(pulse := "pulse_1s", T := #Timers.NC)
      "Time_s"(pulse := "pulse_1s", T := #Timers.SC)
      "Time_s"(pulse := "pulse_1s", T := #Timers.HH)
   END_RUNG
   // the same network as SCL:
   "Time_s"(pulse := "pulse_1s", T := #Timers.NC, ENO => #_w1);
   "Time_s"(EN := #_w1, pulse := "pulse_1s", T := #Timers.SC, ENO => #_w2);
   IF #_w2 THEN "Time_s"(pulse := "pulse_1s", T := #Timers.HH); END_IF;
END_REGION

REGION Network 20: Таймеры, часть 2
   RUNG wire#powerrail
      "Time_s"(pulse := "pulse_1s", T := #Timers.H)
      "Time_s"(pulse := "pulse_1s", T := #Timers.L)
      "Time_s"(pulse := "pulse_1s", T := #Timers.LL)
   END_RUNG
   // the same network as SCL:
   "Time_s"(pulse := "pulse_1s", T := #Timers.H, ENO => #_w1);
   "Time_s"(EN := #_w1, pulse := "pulse_1s", T := #Timers.L, ENO => #_w2);
   IF #_w2 THEN "Time_s"(pulse := "pulse_1s", T := #Timers.LL); END_IF;
END_REGION

REGION Network 21: Сброс сброса
   RUNG wire#powerrail
      Contact( #CMD.Reset )
      R_Coil( #CMD.Reset )
   END_RUNG
   // the same network as SCL:
   IF #CMD.Reset THEN #CMD.Reset := FALSE; END_IF;
END_REGION
END_FUNCTION_BLOCK

FUNCTION_BLOCK "AO_ex"   // FB103, LAD
{ S7_Optimized_Access := 'FALSE' }
VERSION : 0.1
   VAR_INPUT
      SP : Real;   // Уставка авторежима
      All_Block : Bool;   // Аварийная остановка
      pulse : Bool;   // Частота плавного изменения выхода
   END_VAR
   VAR_IN_OUT
      Signal : Int;   // Входной сигнал контроллера
   END_VAR
   VAR
      CMD : Struct   // Основные команды / Блок команд
         Hand : Bool;   // 0 - авто, 1 - ручной / 0 - Авто, 1 - Ручной
         Start_A : Bool := True;   // Автозапуск / Запуск в авторежиме
         Start_M : Bool;   // Ручной - вперёд / Запуск в ручном режиме
         Force : Bool;   // Принудительный
         Lock : Bool;   // Блокировать / Блокировка
         Local : Bool;   // Локальный
         Service : Bool;   // Сервис
         Safety : Bool;   // Безопасность
         Alarm : Bool;   // Есть авария / Авария
         Reset : Bool;   // Сброс аварий
         Sim : Bool;   // Режим симуляции
      END_STRUCT;
      Mode : Int;   // Режим работы
      Status : Int;   // Статус устройства
      Use : Struct   // Функционал
         Inverse : Bool;   // Инвертировать уставку
         Up : Bool;   // Плавный разгон
         Down : Bool;   // Плавный останов
      END_STRUCT;
      Signal_R : Real;   // Актуальный сигнал
      Signal_Ex : Real;   // Конвертация сигнала
      SP_M : Real;   // Уставка в ручном режиме
      Step_up : Real;   // Шаг плавного разгона
      Step_down : Real;   // Шаг плавного останова
      Min_R : Real;   // Минимальная граница
      Max_R : Real;   // Максимальная граница
      Converter : Struct   // Масштабирование сигнала
         Use_Min_In : Bool := true;   // Отсекать входные значения ниже минимума
         Use_Max_In : Bool := true;   // Отсекать входные значения выше максимума
         Use_Min_Out : Bool;   // Отсекать результат ниже минимума
         Use_Max_Out : Bool;   // Отсекать результат выше максимума
         IO : Bool := true;   // Входной/Выходной режим
         Inverse : Bool;   // Инверсия выхода
         Min_In : Real;   // Минимальный входной сигнал
         Max_In : Real := 100.0;   // Максимальный входной сигнал
         Min_Out : Real;   // Минимальный выходной сигнал
         Max_Out : Real := 27648.0;   // Максимальный выходной сигнал
      END_STRUCT;
      T_Up : Struct   // Таймер плавного разгона
         SP : Real;   // Уставка
         Now : Real;   // Текущий счёт
         One : Real := 1.0;   // Вес импульса
         Progress : Real;   // Прогресс выполнения
         "Exit" : Bool;   // Счёт завершён
         Start : Bool;   // Запуск
         Pause : Bool;   // Пауза
         Reset : Bool;   // Сброс счёта
         pos : Bool;   // Контроль фронта сигнала
      END_STRUCT;
      T_Down : Struct   // Таймер плавного останова
         SP : Real;   // Уставка
         Now : Real;   // Текущий счёт
         One : Real := 1.0;   // Вес импульса
         Progress : Real;   // Прогресс выполнения
         "Exit" : Bool;   // Счёт завершён
         Start : Bool;   // Запуск
         Pause : Bool;   // Пауза
         Reset : Bool;   // Сброс счёта
         pos : Bool;   // Контроль фронта сигнала
      END_STRUCT;
   END_VAR
   VAR_TEMP   // added for the SCL form of the ladder/FBD networks
      _w1 : Bool;
   END_VAR
BEGIN

REGION Network 1: Устройство в ручном режиме
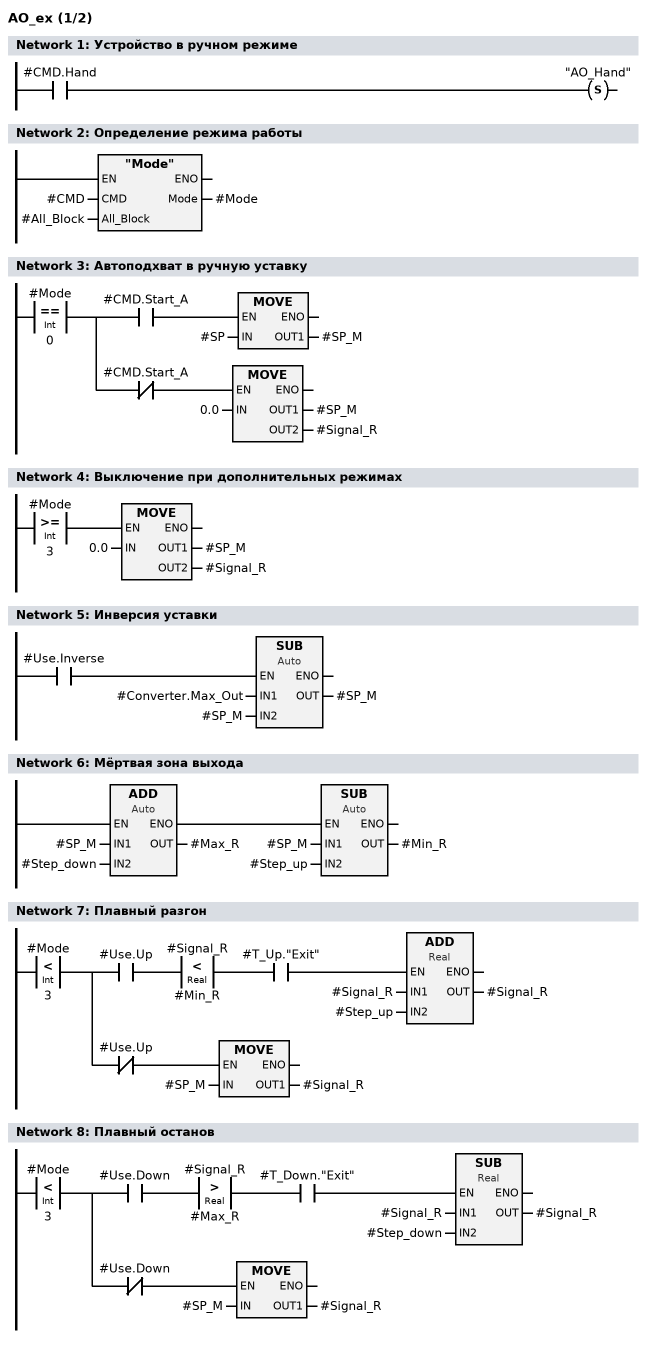
   RUNG wire#powerrail
      Contact( #CMD.Hand )
      S_Coil( "AO_Hand" )
   END_RUNG
   // the same network as SCL:
   IF #CMD.Hand THEN "AO_Hand" := TRUE; END_IF;
END_REGION

REGION Network 2: Определение режима работы
   RUNG wire#powerrail
      "Mode"(CMD := #CMD, All_Block := #All_Block, Mode => #Mode)
   END_RUNG
   // the same network as SCL:
   "Mode"(CMD := #CMD, All_Block := #All_Block, Mode => #Mode);
END_REGION

REGION Network 3: Автоподхват в ручную уставку
   RUNG wire#powerrail
      { S7_Templates := "SrcType := Int" } EQ_Contact(in1 := #Mode, in2 := 0)
      wire#w1
      Contact( #CMD.Start_A )
      { S7_GenerateENO := "TRUE" } Move(in := #SP, out1 => #SP_M)
   END_RUNG
   RUNG wire#w1
      I_Contact( #CMD.Start_A )
      { S7_GenerateENO := "TRUE" } Move(in := 0.0, out1 => #SP_M, out2 => #Signal_R)
   END_RUNG
   // the same network as SCL:
   #_w1 := #Mode = 0;
   IF #_w1 AND #CMD.Start_A THEN #SP_M := #SP; END_IF;
   IF #_w1 AND NOT #CMD.Start_A THEN
       #SP_M := 0.0;
       #Signal_R := 0.0;
   END_IF;
END_REGION

REGION Network 4: Выключение при дополнительных режимах
   RUNG wire#powerrail
      { S7_Templates := "SrcType := Int" } GE_Contact(in1 := #Mode, in2 := 3)
      { S7_GenerateENO := "TRUE" } Move(in := 0.0, out1 => #SP_M, out2 => #Signal_R)
   END_RUNG
   // the same network as SCL:
   IF #Mode >= 3 THEN
       #SP_M := 0.0;
       #Signal_R := 0.0;
   END_IF;
END_REGION

REGION Network 5: Инверсия уставки
   RUNG wire#powerrail
      Contact( #Use.Inverse )
      Sub(in1 := #Converter.Max_Out, in2 := #SP_M, out => #SP_M)
   END_RUNG
   // the same network as SCL:
   IF #Use.Inverse THEN #SP_M := #Converter.Max_Out - #SP_M; END_IF;
END_REGION

REGION Network 6: Мёртвая зона выхода
   RUNG wire#powerrail
      Add(in1 := #SP_M, in2 := #Step_down, out => #Max_R)
      Sub(in1 := #SP_M, in2 := #Step_up, out => #Min_R)
   END_RUNG
   // the same network as SCL:
   #Max_R := #SP_M + #Step_down;
   #Min_R := #SP_M - #Step_up;
END_REGION

REGION Network 7: Плавный разгон
   RUNG wire#powerrail
      { S7_Templates := "SrcType := Int" } LT_Contact(in1 := #Mode, in2 := 3)
      wire#w1
      Contact( #Use.Up )
      { S7_Templates := "SrcType := Real" } LT_Contact(in1 := #Signal_R, in2 := #Min_R)
      Contact( #T_Up."Exit" )
      { S7_Templates := "SrcType := Real"; S7_GenerateENO := "TRUE" } Add(in1 := #Signal_R, in2 := #Step_up, out => #Signal_R)
   END_RUNG
   RUNG wire#w1
      I_Contact( #Use.Up )
      { S7_GenerateENO := "TRUE" } Move(in := #SP_M, out1 => #Signal_R)
   END_RUNG
   // the same network as SCL:
   #_w1 := #Mode < 3;
   IF #_w1 AND #Use.Up AND (#Signal_R < #Min_R) AND #T_Up."Exit" THEN
       #Signal_R := #Signal_R + #Step_up;
   END_IF;
   IF #_w1 AND NOT #Use.Up THEN #Signal_R := #SP_M; END_IF;
END_REGION

REGION Network 8: Плавный останов
   RUNG wire#powerrail
      { S7_Templates := "SrcType := Int" } LT_Contact(in1 := #Mode, in2 := 3)
      wire#w1
      Contact( #Use.Down )
      { S7_Templates := "SrcType := Real" } GT_Contact(in1 := #Signal_R, in2 := #Max_R)
      Contact( #T_Down."Exit" )
      { S7_Templates := "SrcType := Real"; S7_GenerateENO := "TRUE" } Sub(in1 := #Signal_R, in2 := #Step_down, out => #Signal_R)
   END_RUNG
   RUNG wire#w1
      I_Contact( #Use.Down )
      { S7_GenerateENO := "TRUE" } Move(in := #SP_M, out1 => #Signal_R)
   END_RUNG
   // the same network as SCL:
   #_w1 := #Mode < 3;
   IF #_w1 AND #Use.Down AND (#Signal_R > #Max_R) AND #T_Down."Exit" THEN
       #Signal_R := #Signal_R - #Step_down;
   END_IF;
   IF #_w1 AND NOT #Use.Down THEN #Signal_R := #SP_M; END_IF;
END_REGION

REGION Network 9: Масштабирование
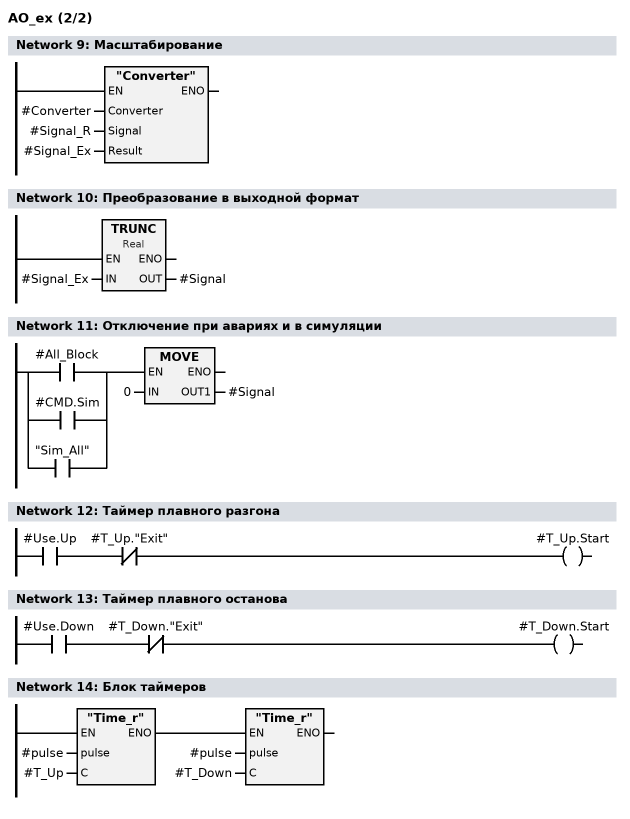
   RUNG wire#powerrail
      "Converter"(Converter := #Converter, Signal := #Signal_R, Result := #Signal_Ex)
   END_RUNG
   // the same network as SCL:
   "Converter"(Converter := #Converter, Signal := #Signal_R, Result := #Signal_Ex);
END_REGION

REGION Network 10: Преобразование в выходной формат
   // no SCL statement known for trunc: written as a call
   trunc(in := #Signal_Ex, out => #Signal);
END_REGION

REGION Network 11: Отключение при авариях и в симуляции
   RUNG wire#powerrail
      Contact( #All_Block )
      wire#w1
      { S7_GenerateENO := "TRUE" } Move(in := 0, out1 => #Signal)
   END_RUNG
   RUNG wire#powerrail
      Contact( #CMD.Sim )
   END_RUNG wire#w1
   RUNG wire#powerrail
      Contact( "Sim_All" )
   END_RUNG wire#w1
   // the same network as SCL:
   IF #All_Block OR #CMD.Sim OR "Sim_All" THEN #Signal := 0; END_IF;
END_REGION

REGION Network 12: Таймер плавного разгона
   RUNG wire#powerrail
      Contact( #Use.Up )
      I_Contact( #T_Up."Exit" )
      Coil( #T_Up.Start )
   END_RUNG
   // the same network as SCL:
   #T_Up.Start := #Use.Up AND NOT #T_Up."Exit";
END_REGION

REGION Network 13: Таймер плавного останова
   RUNG wire#powerrail
      Contact( #Use.Down )
      I_Contact( #T_Down."Exit" )
      Coil( #T_Down.Start )
   END_RUNG
   // the same network as SCL:
   #T_Down.Start := #Use.Down AND NOT #T_Down."Exit";
END_REGION

REGION Network 14: Блок таймеров
   RUNG wire#powerrail
      "Time_r"(pulse := #pulse, C := #T_Up)
      "Time_r"(pulse := #pulse, C := #T_Down)
   END_RUNG
   // the same network as SCL:
   "Time_r"(pulse := #pulse, C := #T_Up, ENO => #_w1);
   IF #_w1 THEN "Time_r"(pulse := #pulse, C := #T_Down); END_IF;
END_REGION
END_FUNCTION_BLOCK

FUNCTION_BLOCK "DRV_Micro"   // FB104, LAD
{ S7_Optimized_Access := 'FALSE' }
VERSION : 0.1
   VAR_INPUT
      Start_A : Bool;   // Запрос запуска
      FB : Bool;   // ОС
      Reset : Bool;   // Сброс аварий
      All_Block : Bool;   // Блокировка
   END_VAR
   VAR_OUTPUT
      CMD : Bool;   // Команда
   END_VAR
   VAR_IN_OUT
      Alarm : Bool;   // Авария
   END_VAR
   VAR
      Hand : Bool;   // Ручной режим
      Start_M : Bool;   // Запуск в ручном режиме
      No_FB : Bool;   // Не использовать ОС
      ON : Bool;   // Успешно запущено
      OFF : Bool;   // Успешно остановлено
      Status : Int;   // Статус устройства / Статус привода
      Wait_On : Struct   // Ожидание ОС контактора / Время на запуск
         SP : Int := 2;
         Now : Int;
         "Exit" : Bool;
         Start : Bool;
         Pause : Bool;
         Reset : Bool;
      END_STRUCT;
      Wait_Off : Struct   // Ожидание концевиков / Время на останов
         SP : Int := 2;
         Now : Int;
         "Exit" : Bool;
         Start : Bool;
         Pause : Bool;
         Reset : Bool;
      END_STRUCT;
   END_VAR
   VAR_TEMP   // added for the SCL form of the ladder/FBD networks
      _w1 : Bool;
      _w2 : Bool;
   END_VAR
BEGIN

REGION Network 1: Управление запуском / дискретный управляющий сигнал
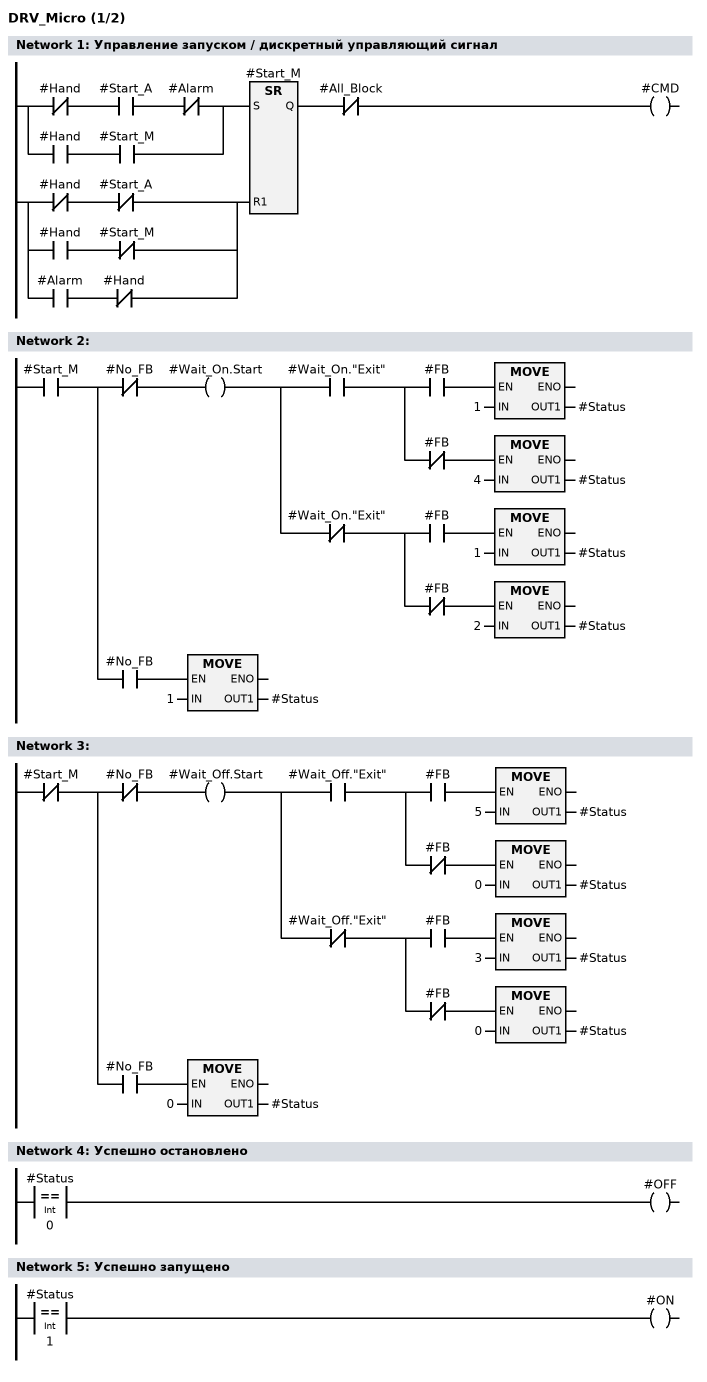
   RUNG wire#powerrail
      I_Contact( #Hand )
      Contact( #Start_A )
      I_Contact( #Alarm )
      wire#w1
      S_SR(operand := #Start_M, r1 := wire#w2)
      I_Contact( #All_Block )
      Coil( #CMD )
   END_RUNG
   RUNG wire#powerrail
      Contact( #Hand )
      Contact( #Start_M )
   END_RUNG wire#w1
   RUNG wire#powerrail
      I_Contact( #Hand )
      I_Contact( #Start_A )
   END_RUNG wire#w2
   RUNG wire#powerrail
      Contact( #Hand )
      I_Contact( #Start_M )
   END_RUNG wire#w2
   RUNG wire#powerrail
      Contact( #Alarm )
      I_Contact( #Hand )
   END_RUNG wire#w2
   // the same network as SCL:
   #_w1 := (NOT #Hand AND NOT #Start_A) OR (#Hand AND NOT #Start_M) OR (#Alarm AND NOT #Hand);
   IF (NOT #Hand AND #Start_A AND NOT #Alarm) OR (#Hand AND #Start_M) THEN
       #Start_M := TRUE;   // SR flip-flop
   END_IF;
   IF #_w1 THEN #Start_M := FALSE; END_IF;
   #CMD := #Start_M AND NOT #All_Block;
END_REGION

REGION Network 2
   RUNG wire#powerrail
      Contact( #Start_M )
      wire#w1
      I_Contact( #No_FB )
      Coil( #Wait_On.Start )
      wire#w2
      Contact( #Wait_On."Exit" )
      wire#w3
      Contact( #FB )
      Move(in := 1, out1 => #Status)
   END_RUNG
   RUNG wire#w3
      I_Contact( #FB )
      Move(in := 4, out1 => #Status)
   END_RUNG
   RUNG wire#w2
      I_Contact( #Wait_On."Exit" )
      wire#w4
      Contact( #FB )
      Move(in := 1, out1 => #Status)
   END_RUNG
   RUNG wire#w4
      I_Contact( #FB )
      Move(in := 2, out1 => #Status)
   END_RUNG
   RUNG wire#w1
      Contact( #No_FB )
      Move(in := 1, out1 => #Status)
   END_RUNG
   // the same network as SCL:
   #Wait_On.Start := #Start_M AND NOT #No_FB;
   #_w1 := #Wait_On.Start AND #Wait_On."Exit";
   IF #_w1 AND #FB THEN #Status := 1; END_IF;
   IF #_w1 AND NOT #FB THEN #Status := 4; END_IF;
   #_w2 := #Wait_On.Start AND NOT #Wait_On."Exit";
   IF #_w2 AND #FB THEN #Status := 1; END_IF;
   IF #_w2 AND NOT #FB THEN #Status := 2; END_IF;
   IF #Start_M AND #No_FB THEN #Status := 1; END_IF;
END_REGION

REGION Network 3
   RUNG wire#powerrail
      I_Contact( #Start_M )
      wire#w1
      I_Contact( #No_FB )
      Coil( #Wait_Off.Start )
      wire#w2
      Contact( #Wait_Off."Exit" )
      wire#w3
      Contact( #FB )
      Move(in := 5, out1 => #Status)
   END_RUNG
   RUNG wire#w3
      I_Contact( #FB )
      Move(in := 0, out1 => #Status)
   END_RUNG
   RUNG wire#w2
      I_Contact( #Wait_Off."Exit" )
      wire#w4
      Contact( #FB )
      Move(in := 3, out1 => #Status)
   END_RUNG
   RUNG wire#w4
      I_Contact( #FB )
      Move(in := 0, out1 => #Status)
   END_RUNG
   RUNG wire#w1
      Contact( #No_FB )
      Move(in := 0, out1 => #Status)
   END_RUNG
   // the same network as SCL:
   #Wait_Off.Start := NOT #Start_M AND NOT #No_FB;
   #_w1 := #Wait_Off.Start AND #Wait_Off."Exit";
   IF #_w1 AND #FB THEN #Status := 5; END_IF;
   IF #_w1 AND NOT #FB THEN #Status := 0; END_IF;
   #_w2 := #Wait_Off.Start AND NOT #Wait_Off."Exit";
   IF #_w2 AND #FB THEN #Status := 3; END_IF;
   IF #_w2 AND NOT #FB THEN #Status := 0; END_IF;
   IF NOT #Start_M AND #No_FB THEN #Status := 0; END_IF;
END_REGION

REGION Network 4: Успешно остановлено
   RUNG wire#powerrail
      { S7_Templates := "SrcType := Int" } EQ_Contact(in1 := #Status, in2 := 0)
      Coil( #OFF )
   END_RUNG
   // the same network as SCL:
   #OFF := #Status = 0;
END_REGION

REGION Network 5: Успешно запущено
   RUNG wire#powerrail
      { S7_Templates := "SrcType := Int" } EQ_Contact(in1 := #Status, in2 := 1)
      Coil( #ON )
   END_RUNG
   // the same network as SCL:
   #ON := #Status = 1;
END_REGION

REGION Network 6: Авария
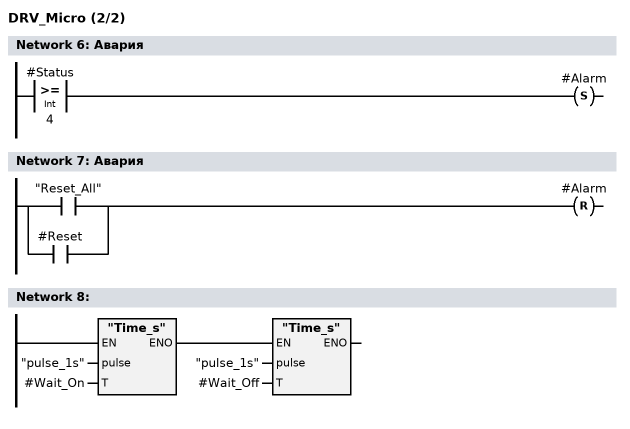
   RUNG wire#powerrail
      { S7_Templates := "SrcType := Int" } GE_Contact(in1 := #Status, in2 := 4)
      S_Coil( #Alarm )
   END_RUNG
   // the same network as SCL:
   IF #Status >= 4 THEN #Alarm := TRUE; END_IF;
END_REGION

REGION Network 7: Авария
   RUNG wire#powerrail
      Contact( "Reset_All" )
      wire#w1
      R_Coil( #Alarm )
   END_RUNG
   RUNG wire#powerrail
      Contact( #Reset )
   END_RUNG wire#w1
   // the same network as SCL:
   IF "Reset_All" OR #Reset THEN #Alarm := FALSE; END_IF;
END_REGION

REGION Network 8
   RUNG wire#powerrail
      "Time_s"(pulse := "pulse_1s", T := #Wait_On)
      "Time_s"(pulse := "pulse_1s", T := #Wait_Off)
   END_RUNG
   // the same network as SCL:
   "Time_s"(pulse := "pulse_1s", T := #Wait_On, ENO => #_w1);
   IF #_w1 THEN "Time_s"(pulse := "pulse_1s", T := #Wait_Off); END_IF;
END_REGION
END_FUNCTION_BLOCK

// folder: Modules

FUNCTION_BLOCK "Motors"   // FB2, LAD
{ S7_Optimized_Access := 'FALSE' }
VERSION : 0.1
   VAR
      T0 : "DRV_M_D";
      T1 : "DRV_M_D";
      T2 : "DRV_M_D";
      T3 : "DRV_M_D";
      T4 : "DRV_M_D";
   END_VAR
   VAR_TEMP   // added for the SCL form of the ladder/FBD networks
      _w1 : Bool;
   END_VAR
   // T0.Use.QF := false;
BEGIN

REGION Network 1
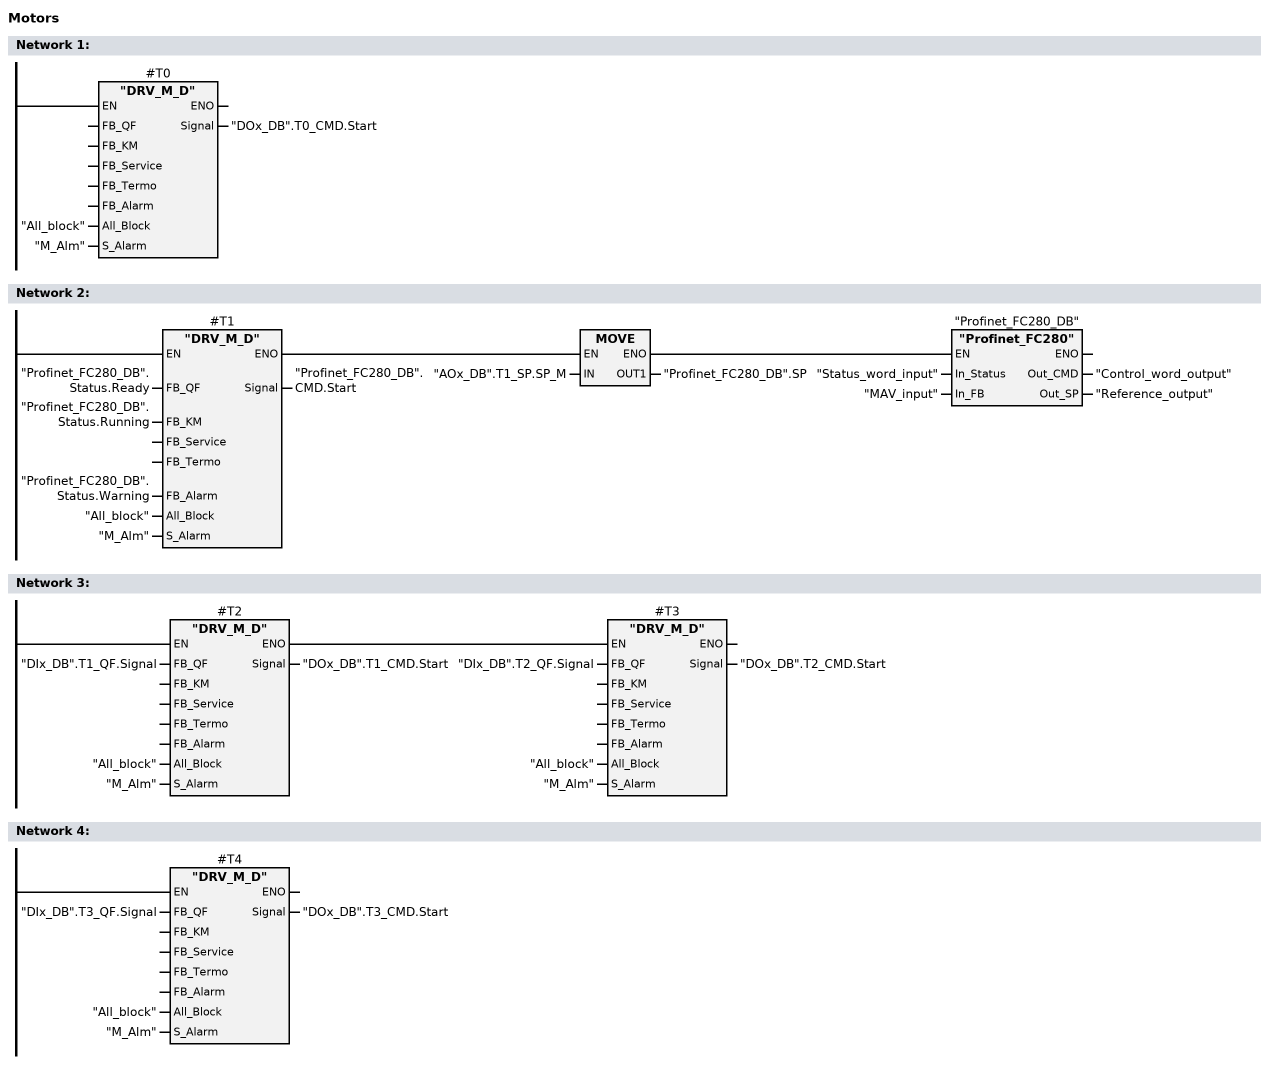
   RUNG wire#powerrail
      #T0(FB_QF :=, FB_KM :=, FB_Service :=, FB_Termo :=, FB_Alarm :=, All_Block := "All_block", S_Alarm := "M_Alm", Signal => "DOx_DB".T0_CMD.Start)
   END_RUNG
   // the same network as SCL:
   #T0(All_Block := "All_block", S_Alarm := "M_Alm", Signal => "DOx_DB".T0_CMD.Start);   // "DRV_M_D"
END_REGION

REGION Network 2
   RUNG wire#powerrail
      #T1(FB_QF := "Profinet_FC280_DB".Status.Ready, FB_KM := "Profinet_FC280_DB".Status.Running, FB_Service :=, FB_Termo :=, FB_Alarm := "Profinet_FC280_DB".Status.Warning, All_Block := "All_block", S_Alarm := "M_Alm", Signal => "Profinet_FC280_DB".CMD.Start)
      Move(in := "AOx_DB".T1_SP.SP_M, out1 => "Profinet_FC280_DB".SP)
      "Profinet_FC280_DB"(In_Status := "Status_word_input", In_FB := "MAV_input", Out_CMD => "Control_word_output", Out_SP => "Reference_output")
   END_RUNG
   // the same network as SCL:
   #T1(FB_QF := "Profinet_FC280_DB".Status.Ready,   // "DRV_M_D"
       FB_KM := "Profinet_FC280_DB".Status.Running,
       FB_Alarm := "Profinet_FC280_DB".Status.Warning,
       All_Block := "All_block",
       S_Alarm := "M_Alm",
       Signal => "Profinet_FC280_DB".CMD.Start,
       ENO => #_w1);
   IF #_w1 THEN
       "Profinet_FC280_DB".SP := "AOx_DB".T1_SP.SP_M;
       "Profinet_FC280_DB"(In_Status := "Status_word_input",   // "Profinet_FC280"
                           In_FB := "MAV_input",
                           Out_CMD => "Control_word_output",
                           Out_SP => "Reference_output");
   END_IF;
END_REGION

REGION Network 3
   RUNG wire#powerrail
      #T2(FB_QF := "DIx_DB".T1_QF.Signal, FB_KM :=, FB_Service :=, FB_Termo :=, FB_Alarm :=, All_Block := "All_block", S_Alarm := "M_Alm", Signal => "DOx_DB".T1_CMD.Start)
      #T3(FB_QF := "DIx_DB".T2_QF.Signal, FB_KM :=, FB_Service :=, FB_Termo :=, FB_Alarm :=, All_Block := "All_block", S_Alarm := "M_Alm", Signal => "DOx_DB".T2_CMD.Start)
   END_RUNG
   // the same network as SCL:
   #T2(FB_QF := "DIx_DB".T1_QF.Signal,   // "DRV_M_D"
       All_Block := "All_block",
       S_Alarm := "M_Alm",
       Signal => "DOx_DB".T1_CMD.Start,
       ENO => #_w1);
   IF #_w1 THEN
       #T3(FB_QF := "DIx_DB".T2_QF.Signal,   // "DRV_M_D"
           All_Block := "All_block",
           S_Alarm := "M_Alm",
           Signal => "DOx_DB".T2_CMD.Start);
   END_IF;
END_REGION

REGION Network 4
   RUNG wire#powerrail
      #T4(FB_QF := "DIx_DB".T3_QF.Signal, FB_KM :=, FB_Service :=, FB_Termo :=, FB_Alarm :=, All_Block := "All_block", S_Alarm := "M_Alm", Signal => "DOx_DB".T3_CMD.Start)
   END_RUNG
   // the same network as SCL:
   #T4(FB_QF := "DIx_DB".T3_QF.Signal,   // "DRV_M_D"
       All_Block := "All_block",
       S_Alarm := "M_Alm",
       Signal => "DOx_DB".T3_CMD.Start);
END_REGION
END_FUNCTION_BLOCK

FUNCTION_BLOCK "Valves"   // FB3, LAD
{ S7_Optimized_Access := 'FALSE' }
VERSION : 0.1
   VAR
      V1 : "DRV_V_D2";
      V2 : "DRV_V_D2";
      V3 : "DRV_V_D2";
   END_VAR
   VAR_TEMP   // added for the SCL form of the ladder/FBD networks
      _w1 : Bool;
      _w2 : Bool;
   END_VAR
   // V1.Use.KM_Open := false;
   // V1.Use.Close := true;
   // V1.Use.Open := false;
   // V2.Use.KM_Open := false;
   // V2.Use.Close := true;
   // V3.Use.KM_Open := false;
   // V3.Use.Close := true;
BEGIN

REGION Network 1
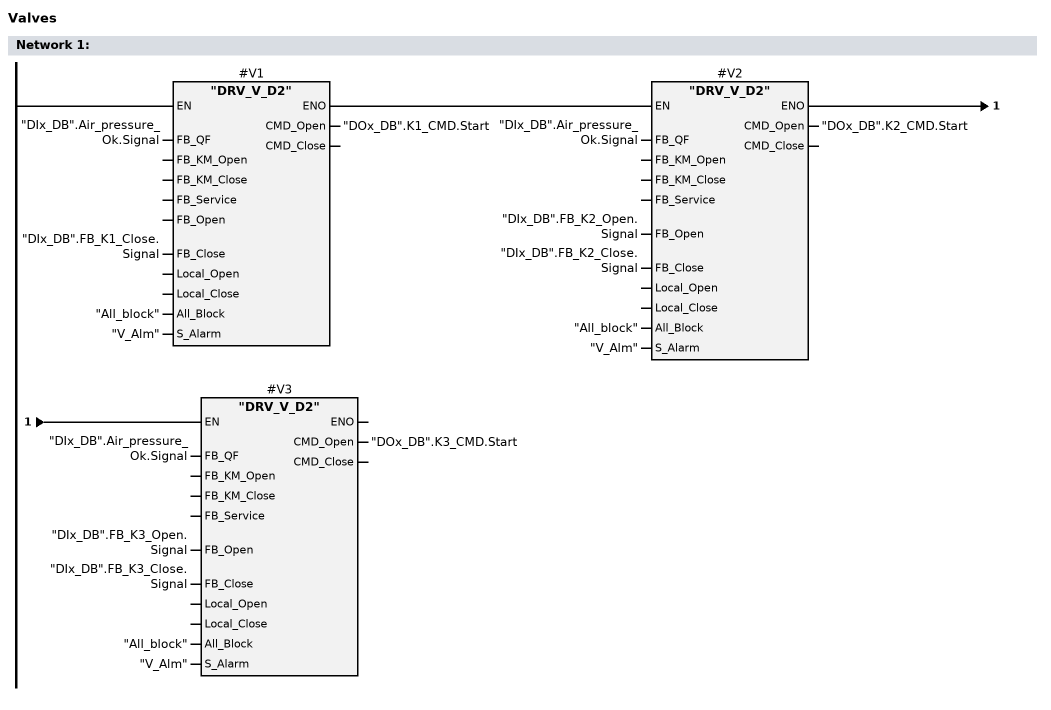
   RUNG wire#powerrail
      #V1(FB_QF := "DIx_DB".Air_pressure_Ok.Signal, FB_KM_Open :=, FB_KM_Close :=, FB_Service :=, FB_Open :=, FB_Close := "DIx_DB".FB_K1_Close.Signal, Local_Open :=, Local_Close :=, All_Block := "All_block", S_Alarm := "V_Alm", CMD_Open => "DOx_DB".K1_CMD.Start, CMD_Close =>)
      #V2(FB_QF := "DIx_DB".Air_pressure_Ok.Signal, FB_KM_Open :=, FB_KM_Close :=, FB_Service :=, FB_Open := "DIx_DB".FB_K2_Open.Signal, FB_Close := "DIx_DB".FB_K2_Close.Signal, Local_Open :=, Local_Close :=, All_Block := "All_block", S_Alarm := "V_Alm", CMD_Open => "DOx_DB".K2_CMD.Start, CMD_Close =>)
      #V3(FB_QF := "DIx_DB".Air_pressure_Ok.Signal, FB_KM_Open :=, FB_KM_Close :=, FB_Service :=, FB_Open := "DIx_DB".FB_K3_Open.Signal, FB_Close := "DIx_DB".FB_K3_Close.Signal, Local_Open :=, Local_Close :=, All_Block := "All_block", S_Alarm := "V_Alm", CMD_Open => "DOx_DB".K3_CMD.Start, CMD_Close =>)
   END_RUNG
   // the same network as SCL:
   #V1(FB_QF := "DIx_DB".Air_pressure_Ok.Signal,   // "DRV_V_D2"
       FB_Close := "DIx_DB".FB_K1_Close.Signal,
       All_Block := "All_block",
       S_Alarm := "V_Alm",
       CMD_Open => "DOx_DB".K1_CMD.Start,
       ENO => #_w1);
   #V2(EN := #_w1,   // "DRV_V_D2"
       FB_QF := "DIx_DB".Air_pressure_Ok.Signal,
       FB_Open := "DIx_DB".FB_K2_Open.Signal,
       FB_Close := "DIx_DB".FB_K2_Close.Signal,
       All_Block := "All_block",
       S_Alarm := "V_Alm",
       CMD_Open => "DOx_DB".K2_CMD.Start,
       ENO => #_w2);
   IF #_w2 THEN
       #V3(FB_QF := "DIx_DB".Air_pressure_Ok.Signal,   // "DRV_V_D2"
           FB_Open := "DIx_DB".FB_K3_Open.Signal,
           FB_Close := "DIx_DB".FB_K3_Close.Signal,
           All_Block := "All_block",
           S_Alarm := "V_Alm",
           CMD_Open => "DOx_DB".K3_CMD.Start);
   END_IF;
END_REGION
END_FUNCTION_BLOCK

FUNCTION_BLOCK "AOx"   // FB7, LAD
{ S7_Optimized_Access := 'FALSE' }
VERSION : 0.1
   VAR
      T1_SP : "AO_ex";
   END_VAR
BEGIN

REGION Network 1
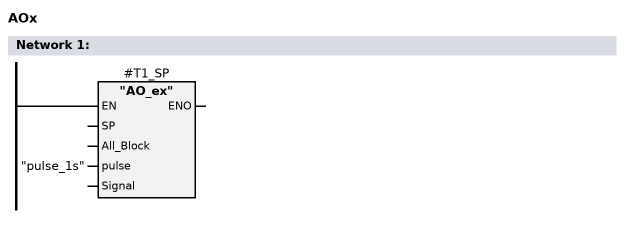
   RUNG wire#powerrail
      #T1_SP(SP :=, All_Block :=, pulse := "pulse_1s", Signal :=)
   END_RUNG
   // the same network as SCL:
   #T1_SP(pulse := "pulse_1s");   // "AO_ex"
END_REGION
END_FUNCTION_BLOCK

FUNCTION_BLOCK "DIx"   // FB8, LAD
{ S7_Optimized_Access := 'FALSE' }
VERSION : 0.1
   VAR
      Voltage_CPU_Ok : "DI_ex";
      Voltage_DI_Ok : "DI_ex";
      Voltage_DO_Ok : "DI_ex";
      Voltage_24V_Ok : "DI_ex";
      Safety_Ok : "DI_ex";
      Cold_tunnel_QF : "DI_ex";
      T1_QF : "DI_ex";
      T2_QF : "DI_ex";
      T3_QF : "DI_ex";
      T1_Box_ready : "DI_ex";
      T2_Box_Ready : "DI_ex";
      T3_Box_Ready : "DI_ex";
      Air_pressure_Ok : "DI_ex";
      FB_K1_Close : "DI_ex";
      FB_K2_Open : "DI_ex";
      FB_K2_Close : "DI_ex";
      FB_K3_Open : "DI_ex";
      FB_K3_Close : "DI_ex";
   END_VAR
   VAR_TEMP   // added for the SCL form of the ladder/FBD networks
      _w1 : Bool;
      _w2 : Bool;
      _w3 : Bool;
      _w4 : Bool;
   END_VAR
BEGIN

REGION Network 1
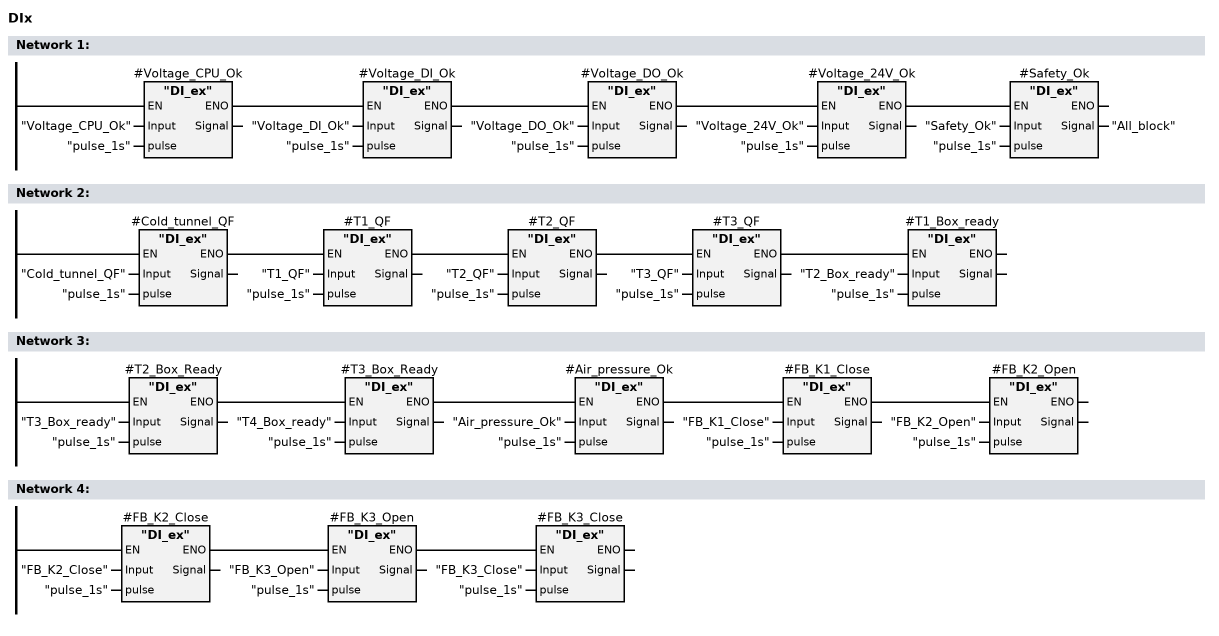
   RUNG wire#powerrail
      #Voltage_CPU_Ok(Input := "Voltage_CPU_Ok", pulse := "pulse_1s", Signal =>)
      #Voltage_DI_Ok(Input := "Voltage_DI_Ok", pulse := "pulse_1s", Signal =>)
      #Voltage_DO_Ok(Input := "Voltage_DO_Ok", pulse := "pulse_1s", Signal =>)
      #Voltage_24V_Ok(Input := "Voltage_24V_Ok", pulse := "pulse_1s", Signal =>)
      #Safety_Ok(Input := "Safety_Ok", pulse := "pulse_1s", Signal => "All_block")
   END_RUNG
   // the same network as SCL:
   #Voltage_CPU_Ok(Input := "Voltage_CPU_Ok", pulse := "pulse_1s", ENO => #_w1);   // "DI_ex"
   #Voltage_DI_Ok(EN := #_w1, Input := "Voltage_DI_Ok", pulse := "pulse_1s", ENO => #_w2);   // "DI_ex"
   #Voltage_DO_Ok(EN := #_w2, Input := "Voltage_DO_Ok", pulse := "pulse_1s", ENO => #_w3);   // "DI_ex"
   #Voltage_24V_Ok(EN := #_w3, Input := "Voltage_24V_Ok", pulse := "pulse_1s", ENO => #_w4);   // "DI_ex"
   IF #_w4 THEN
       #Safety_Ok(Input := "Safety_Ok", pulse := "pulse_1s", Signal => "All_block");   // "DI_ex"
   END_IF;
END_REGION

REGION Network 2
   RUNG wire#powerrail
      #Cold_tunnel_QF(Input := "Cold_tunnel_QF", pulse := "pulse_1s", Signal =>)
      #T1_QF(Input := "T1_QF", pulse := "pulse_1s", Signal =>)
      #T2_QF(Input := "T2_QF", pulse := "pulse_1s", Signal =>)
      #T3_QF(Input := "T3_QF", pulse := "pulse_1s", Signal =>)
      #T1_Box_ready(Input := "T2_Box_ready", pulse := "pulse_1s", Signal =>)
   END_RUNG
   // the same network as SCL:
   #Cold_tunnel_QF(Input := "Cold_tunnel_QF", pulse := "pulse_1s", ENO => #_w1);   // "DI_ex"
   #T1_QF(EN := #_w1, Input := "T1_QF", pulse := "pulse_1s", ENO => #_w2);   // "DI_ex"
   #T2_QF(EN := #_w2, Input := "T2_QF", pulse := "pulse_1s", ENO => #_w3);   // "DI_ex"
   #T3_QF(EN := #_w3, Input := "T3_QF", pulse := "pulse_1s", ENO => #_w4);   // "DI_ex"
   IF #_w4 THEN
       #T1_Box_ready(Input := "T2_Box_ready", pulse := "pulse_1s");   // "DI_ex"
   END_IF;
END_REGION

REGION Network 3
   RUNG wire#powerrail
      #T2_Box_Ready(Input := "T3_Box_ready", pulse := "pulse_1s", Signal =>)
      #T3_Box_Ready(Input := "T4_Box_ready", pulse := "pulse_1s", Signal =>)
      #Air_pressure_Ok(Input := "Air_pressure_Ok", pulse := "pulse_1s", Signal =>)
      #FB_K1_Close(Input := "FB_K1_Close", pulse := "pulse_1s", Signal =>)
      #FB_K2_Open(Input := "FB_K2_Open", pulse := "pulse_1s", Signal =>)
   END_RUNG
   // the same network as SCL:
   #T2_Box_Ready(Input := "T3_Box_ready", pulse := "pulse_1s", ENO => #_w1);   // "DI_ex"
   #T3_Box_Ready(EN := #_w1, Input := "T4_Box_ready", pulse := "pulse_1s", ENO => #_w2);   // "DI_ex"
   #Air_pressure_Ok(EN := #_w2, Input := "Air_pressure_Ok", pulse := "pulse_1s", ENO => #_w3);   // "DI_ex"
   #FB_K1_Close(EN := #_w3, Input := "FB_K1_Close", pulse := "pulse_1s", ENO => #_w4);   // "DI_ex"
   IF #_w4 THEN
       #FB_K2_Open(Input := "FB_K2_Open", pulse := "pulse_1s");   // "DI_ex"
   END_IF;
END_REGION

REGION Network 4
   RUNG wire#powerrail
      #FB_K2_Close(Input := "FB_K2_Close", pulse := "pulse_1s", Signal =>)
      #FB_K3_Open(Input := "FB_K3_Open", pulse := "pulse_1s", Signal =>)
      #FB_K3_Close(Input := "FB_K3_Close", pulse := "pulse_1s", Signal =>)
   END_RUNG
   // the same network as SCL:
   #FB_K2_Close(Input := "FB_K2_Close", pulse := "pulse_1s", ENO => #_w1);   // "DI_ex"
   #FB_K3_Open(EN := #_w1, Input := "FB_K3_Open", pulse := "pulse_1s", ENO => #_w2);   // "DI_ex"
   IF #_w2 THEN
       #FB_K3_Close(Input := "FB_K3_Close", pulse := "pulse_1s");   // "DI_ex"
   END_IF;
END_REGION
END_FUNCTION_BLOCK

FUNCTION_BLOCK "DOx"   // FB9, LAD
{ S7_Optimized_Access := 'FALSE' }
VERSION : 0.1
   VAR
      T0_CMD : "DO_ex";
      T1_CMD : "DO_ex";
      T2_CMD : "DO_ex";
      T3_CMD : "DO_ex";
      K1_CMD : "DO_ex";
      K2_CMD : "DO_ex";
      K3_CMD : "DO_ex";
      Supply_allowed : "DO_ex";
      Reset_Safety : "DO_ex";
      Reset : "DO_ex";
      Green : "DO_ex";
      Red : "DO_ex";
      Blue : "DO_ex";
      Orange : "DO_ex";
   END_VAR
   VAR_TEMP   // added for the SCL form of the ladder/FBD networks
      _w1 : Bool;
      _w2 : Bool;
      _w3 : Bool;
   END_VAR
BEGIN

REGION Network 1
